// TwinCAT 3 PLC project ICPPLC
// ProgramVersion: 3.1.4023.0
// CompilerDefines: VISU_USEWSTRING
// libraries:
//   Tc2_Math, * (Beckhoff Automation GmbH)
//   Tc2_MC2, * (Beckhoff Automation GmbH)
//   Tc2_SerialCom, * (Beckhoff Automation GmbH)
//   Tc2_Standard, * (Beckhoff Automation GmbH)
//   Tc2_SUPS, * (Beckhoff Automation GmbH)
//   Tc2_System, * (Beckhoff Automation GmbH)
//   Tc2_TcpIp, * (Beckhoff Automation GmbH)
//   Tc2_Utilities, * (Beckhoff Automation GmbH)
//   Tc3_Module, * (Beckhoff Automation GmbH)
//   VisuDialogs, * (System)
//   VisuSymbols, * (System)
// project tree:
//   / ComTask.TcTTO, DataSave_1.TcTTO, GlobalTextList.TcGTLO, IOTask.TcTTO, PlcTask.TcTTO, VISU_TASK.TcTTO, 视图管理器.TcVMO (not stored)
//   DUTs/ ST_A2BData.TcDUT, ST_B2AData.TcDUT
//   GVLs/ GVL_AllCONSTANT.TcGVL, GVL_AllGLOBAL.TcGVL, GVL_AllPERSISTENT.TcGVL, GVL_Datasave.TcGVL
//   POUs/BaseModule/ActionModule/ARMModule/ ARMModule.TcPOU
//   POUs/BaseModule/ActionModule/ARMModule/enum/ ARMType.TcDUT
//   POUs/BaseModule/ActionModule/ARMModule/struct/ ARMModuleHMI.TcDUT
//   POUs/BaseModule/ActionModule/cylinderModule/ CylinderModule.TcPOU
//   POUs/BaseModule/ActionModule/cylinderModule/enum/ CylinderType.TcDUT
//   POUs/BaseModule/ActionModule/cylinderModule/struct/ cylinderModuleHMI.TcDUT
//   POUs/BaseModule/ActionModule/cylinderModule/visu/ cylinderModuleVisu.TcVIS, cylinderModuleVisu_1.TcVIS
//   POUs/BaseModule/ActionModule/chillerModule/ ChillerModule_1.TcPOU
//   POUs/BaseModule/ActionModule/chillerModule/enum/ chillerType.TcDUT
//   POUs/BaseModule/ActionModule/chillerModule/struct/ chillerModuleHMI.TcDUT
//   POUs/BaseModule/ActionModule/enum/ ControlMode.TcDUT
//   POUs/BaseModule/ActionModule/ GVL_ActionModule.TcGVL
//   POUs/BaseModule/ActionModule/HEATModule/enum/ HEATType.TcDUT
//   POUs/BaseModule/ActionModule/HEATModule/ HeatModule.TcPOU
//   POUs/BaseModule/ActionModule/HEATModule/struct/ HEATModuleHMI.TcDUT
//   POUs/BaseModule/ActionModule/HEATModule/visu/ HeatModuleVisu.TcVIS
//   POUs/BaseModule/ActionModule/MFCModule/enum/ MFCType.TcDUT
//   POUs/BaseModule/ActionModule/MFCModule/ MFCModule.TcPOU
//   POUs/BaseModule/ActionModule/MFCModule/struct/ MFCStruct.TcDUT
//   POUs/BaseModule/ActionModule/motorModule/enum/ MotorHomeMode.TcDUT, MotorType.TcDUT
//   POUs/BaseModule/ActionModule/motorModule/ FB_MotorMovements.TcPOU, MotionModule.TcPOU
//   POUs/BaseModule/ActionModule/motorModule/struct/ motionModuleDataHMI.TcDUT, ST_MotorOutput.TcDUT
//   POUs/BaseModule/ActionModule/motorModule/visu/ motionModuleP1.TcVIS, motionModuleP2.TcVIS, motionModuleP3.TcVIS
//   POUs/BaseModule/ActionModule/OtherModule/ ChillerModule.TcPOU, GaugeViewModule.TcPOU, ChamberGaugeViewModule.TcPOU
//   POUs/BaseModule/ActionModule/PendulumValveModule/enum/ PVControlMOD.TcDUT, PVType.TcDUT
//   POUs/BaseModule/ActionModule/PendulumValveModule/ PVModule.TcPOU
//   POUs/BaseModule/ActionModule/PendulumValveModule/struct/ PVModuleHMI.TcDUT
//   POUs/BaseModule/ActionModule/RFModule/enum/ RFType.TcDUT
//   POUs/BaseModule/ActionModule/RFModule/ RFModule.TcPOU
//   POUs/BaseModule/ActionModule/RFModule/struct/ RFHMIStruts.TcDUT
//   POUs/BaseModule/ActionModule/RFModule_Source/ RFModule_Source.TcPOU
//   POUs/BaseModule/ActionModule/TMPModule/enum/ TMPType.TcDUT
//   POUs/BaseModule/ActionModule/TMPModule/struct/ TMPHMIStruts.TcDUT
//   POUs/BaseModule/ActionModule/TMPModule/ TMPModule.TcPOU
//   POUs/BaseModule/ActionModule/TMPModule/visu/ TMPModuleVisu.TcVIS
//   POUs/BaseModule/ActionModule/VPEModule/enum/ VPEType.TcDUT
//   POUs/BaseModule/ActionModule/VPEModule/struct/ VPEHMIStruts.TcDUT, VPETestStruts530.TcDUT, VPETestStruts540.TcDUT
//   POUs/BaseModule/ActionModule/VPEModule/visu/ VPEModuleVis.TcVIS
//   POUs/BaseModule/ActionModule/VPEModule/ VPEModule.TcPOU
//   POUs/BaseModule/COE/ EcCoeSdo_ForTest.TcPOU, FB_ECCOE_READ_WRITE.TcPOU
//   POUs/BaseModule/Communication/ FuncModule_RS232_Byte.TcPOU, FuncModule_RS232_SRF.TcPOU, FuncModule_RS232_ARM.TcPOU, FuncModule_RS485_MFC.TcPOU, FuncModule_RS232_TBP.TcPOU, FuncModule_TCPIP_Binary_POU.TcPOU, FuncModule_TCPIP_String_POU.TcPOU
//   POUs/BaseModule/Communication/struct/ struct_byte_1.TcDUT, struct_Tester.TcDUT, struct_byte.TcDUT
//   POUs/BaseModule/DataSaveModule_EX/csvReadWriteInTextMode/ P_TextModeDelete_1.TcPOU, P_TextModeRead.TcPOU, P_TextModeRead_Recipe.TcPOU, P_TextModeRead_RecipeName.TcPOU, P_TextModeWrite.TcPOU, P_TextModeWrite_Recipe.TcPOU, P_TextModeWrite_RecipeName.TcPOU, StringModel_256000_EX.TcPOU
//   POUs/BaseModule/DataSaveModule_EX/ DataSaveModule_EX.TcPOU, GVL_DataSave_EX.TcGVL, RecipeNameModule_EX.TcPOU, RecipeSaveModule_EX.TcPOU
//   POUs/BaseModule/DataSaveModule_EX/Struct/ RecipeNamePar.TcDUT, RecipePar.TcDUT, RecipeShowStr.TcDUT
//   POUs/BaseModule/EL2252_2262Control/ FlipperModule_EL2252.TcPOU, FlipperModule_EL2262.TcPOU, FlipperModule_EL2262_old.TcPOU
//   POUs/BaseModule/EL2252_2262Control/SquareWaveOut/ FB_SquareWaveOut_EL2262.TcPOU, SquareWaveOut_EL2262_TEST.TcPOU
//   POUs/BaseModule/EL2252_2262Control/struct/ ST_CamSwitch.TcDUT, ST_CamSwitch_EL2262.TcDUT, ST_EL2262OutData.TcDUT
//   POUs/BaseModule/Error/enum/ Error_Level.TcDUT
//   POUs/BaseModule/Error/ ErrCodeProcess.TcPOU, errorMonitor.TcPOU, error_Printf.TcPOU, error_Trigger.TcPOU, GVL_Error.TcGVL
//   POUs/BaseModule/Error/struct/ ST_Error.TcDUT
//   POUs/BaseModule/IO/ FB_IOBase_Input_New.TcPOU, FB_IOBase_Output_New.TcPOU
//   POUs/BaseModule/IO/ReadWriteCSV/ FB_IOFileReadWrite.TcPOU, POU_Test.TcPOU, ST_DataFmtBase.TcDUT
//   POUs/BaseModule/IO/struct/ ST_INPUT_IO.TcDUT, ST_IOBase_Show_HMI.TcDUT, ST_OUTPUT_IO.TcDUT
//   POUs/BaseModule/IO/visu/ IOBase_Show_New.TcVIS
//   POUs/BaseModule/MainFrame/ MainFram.TcDUT, MainFrame.TcVIS
//   POUs/BaseModule/PrintLogModule_EX/ GVL_PrintLogModule_EX.TcGVL, printLogModule_EX.TcPOU
//   POUs/BaseModule/PrintLogModule_EX/struct/ printLogModule_EX_DataHMI.TcDUT, printLogModule_EX_DataST.TcDUT, ST_DeleteFile.TcDUT
//   POUs/BaseModule/PrintLogModule_EX/visu/ showInfo_Auto.TcVIS, showInfo.TcVIS
//   POUs/BaseModule/SystemTimeModule/ GVL_SystemTimeModule.TcGVL, systemTimeModule.TcPOU
//   POUs/BaseModule/TcpIpModule_EX/ ALCData2String.TcPOU, CloseAllSocket.TcPOU, GVL_TcpIpModule_EX.TcGVL
//   POUs/BaseModule/TcpIpModule_EX/clientModule_EX/ tcpipClientModule_EX.TcPOU
//   POUs/BaseModule/TcpIpModule_EX/dataStruct_EX/ ST_TCPIP_DATA_STRUCT_ALC.TcDUT
//   POUs/BaseModule/TcpIpModule_EX/serverModule_EX/ tcpipServerModule_EX.TcPOU
//   POUs/BaseModule/UPS_CX51X0/ ups_CX51X0.TcPOU
//   POUs/Communication/ Communication_Error.TcPOU, PLC_Chiller.TcPOU, PLC_AMX_AI.TcPOU, PLC_FreeByte.TcPOU, PLC_PDV.TcPOU, PLC_HeliumPressure.TcPOU, PLC_SourceRF.TcPOU, PLC_PowerRF.TcPOU, PRG_ADS_Comm_ByName_A2B.TcPOU, RS232_485_ALLEL.TcPOU, PLC_String.TcPOU, PLC_SW1.TcPOU, ServicesRefreshPOU.TcPOU
//   POUs/Communication/Communica_ALC/ enum_CommandNumber.TcDUT, E_Sta1_CMD.TcDUT
//   POUs/Data/ DataSave.TcPOU, DownTimeRecordPOU.TcPOU, FB_SavePar.TcPOU, FB_WStringSave.TcPOU, Test_FilePOU.TcPOU
//   POUs/Instance/ instance.TcPOU, InstanceUtility.TcPOU
//   POUs/IO/ TesterIO.TcPOU
//   POUs/MachinePOU/SemiAutomatic/ S_BackOfHeliumClear.TcPOU, S_CO_ControlRF.TcPOU, S_PDVSafeCtr.TcPOU, S_MachineVent.TcPOU, S_Etching.TcPOU, S_LoadLockPumping.TcPOU, S_LoadLockVent.TcPOU, S_ChamberLLVent.TcPOU, S_MachinePumping.TcPOU, S_UnLoadWafer.TcPOU, S_WaferCheckPOU.TcPOU, S_RoughPumping.TcPOU, S_ActuatorRecoveryPOU.TcPOU, S_LoadWafer.TcPOU
//   POUs/MachinePOU/State/ otherMachineState.TcPOU
//   POUs/MachinePOU/ MainPOU.TcPOU
//   POUs/ MAIN.TcPOU
//   POUs/Other/ActBase/ ActStepBase.TcPOU
//   POUs/Other/ActBase/ITF/ ITFActStep.TcIO, ITFUserAction.TcIO
//   POUs/Other/ActBase/ITF/struct/ ST_ActStep_State.TcDUT
//   POUs/Other/HMI/ Note.TcVIS, WARMStruct.TcDUT, WARM.TcVIS, NoteStruct.TcDUT
//   POUs/Other/MachineState/enum/ RunningStatus.TcDUT
//   POUs/Other/MachineState/ FB_MachineState.TcPOU, GVL_MachineState.TcGVL, MachineStatePOU.TcPOU, MainParComfer_HMI.TcPOU, ST_DownTimeRecord.TcDUT, ST_MachineState.TcDUT
//   POUs/Other/ MainRunPOU.TcPOU
//   POUs/Other/Struct/ActPos/ ST_DOEActPos.TcDUT
//   POUs/Other/Struct/StationBuild/ ST_ICP.TcDUT
//   POUs/Other/Struct/ ST_HaveDUTState.TcDUT, ST_MachineUtility.TcDUT, ST_POUCommunication.TcDUT, ST_StationConfigBase.TcDUT
//   VISUs/Editor/ Manual.TcVIS, Overview.TcVIS, Overview_Total.TcVIS, ViewPar.TcVIS, ViewPar_1.TcVIS
//   VISUs/Config/ Config.TcVIS, Config_Base.TcVIS
//   VISUs/ ImagePool1.TcIPO (not stored), Loadding.TcVIS, Main.TcVIS
//   VISUs/IO/ IO.TcVIS, IO_Input.TcVIS, IO_Output.TcVIS
//   VISUs/Log/ LogInf.TcVIS
//   VISUs/Operator/ Operator.TcVIS
//   VISUs/Recipe/ Recipe.TcVIS, Recipe_Operator.TcVIS
//   VISUs/TextList/ CtrlModeTextList.TcTLO, MachineStateTextList.TcTLO, PDVConfigMode.TcTLO, RunModeTypeTexList.TcTLO
// real-time tasks:
//   TASK PlcTask: cycle T#10ms, priority 17, ADS port 350
//   TASK VISU_TASK: cycle T#100000us, priority 30, ADS port 351
//   TASK DataSave_1: cycle T#20ms, priority 18, ADS port 352
//   TASK IOTask: cycle T#2ms, priority 12, ADS port 353
//   TASK ComTask: cycle T#2ms, priority 19, ADS port 354
// I/O:
//   DEVICE Device 1 (EtherCAT), AmsNetId 5.114.113.208.2.1
//     Term 1 (EK1200) [EK1200-5000 EtherCAT Power supply (2A E-Bus)]
//       Term 2 (EL1889) [EL1889 16Ch. Dig. Input 24V, 3ms, negative]
//       Term 3 (EL1889) [EL1889 16Ch. Dig. Input 24V, 3ms, negative]
//       Term 4 (EL2889) [EL2889 16Ch. Dig. Output 24V, 0.5A, negative]
//       Term 5 (EL2889) [EL2889 16Ch. Dig. Output 24V, 0.5A, negative]
//       Term 6 (EL2889) [EL2889 16Ch. Dig. Output 24V, 0.5A, negative]
//       Term 7 (EL3174) [EL3174 4K. Ana. Eingang  +/-10V Diff., +/-20mA SingleEnded, 16 Bit]
//       Term 8 (EL6002) [EL6002 Interface 2Ch. (RS232)]
//       Term 9 (EL6002) [EL6002 Interface 2Ch. (RS232)]
//       Term 10 (EL6022) [EL6022 Interface 2Ch. (RS422/485)]
//       Term 11 (EK1110) [EK1110 EtherCAT extension]
//   DEVICE Device 6 (EtherCAT), AmsNetId 5.114.113.208.7.1
//     Box 12 (EC SERIES) [EC SERIES]
// variable links:
//   ICPPLC/ICPPLC Instance <-> Device 1 (EtherCAT)/Term 1 (EK1200)/Term 10 (EL6022)
//     ComTask Inputs/RS232_485_ALLEL.MFC_COMin/D[{0..21}] <-> COM Inputs Channel 2/Data In {0..21}  (22 links)
//     ComTask Inputs/RS232_485_ALLEL.MFC_COMin/Status <-> COM Inputs Channel 2/Status
//     ComTask Outputs/RS232_485_ALLEL.MFC_COMout/Ctrl <-> COM Outputs Channel 2/Ctrl
//     ComTask Outputs/RS232_485_ALLEL.MFC_COMout/D[{0..21}] <-> COM Outputs Channel 2/Data Out {0..21}  (22 links)
//   ICPPLC/ICPPLC Instance <-> Device 1 (EtherCAT)/Term 1 (EK1200)/Term 2 (EL1889)
//     IOTask Inputs/TesterIO.fbIOBase_Input.stIOBase[1].io[{1..16}] <-> Channel {1..16}/Input  (16 links)
//   ICPPLC/ICPPLC Instance <-> Device 1 (EtherCAT)/Term 1 (EK1200)/Term 3 (EL1889)
//     IOTask Inputs/TesterIO.fbIOBase_Input.stIOBase[2].io[{1..16}] <-> Channel {1..16}/Input  (16 links)
//   ICPPLC/ICPPLC Instance <-> Device 1 (EtherCAT)/Term 1 (EK1200)/Term 4 (EL2889)
//     IOTask Outputs/TesterIO.fbIOBase_Output.stIOBase[1].io[{1..16}] <-> Channel {1..16}/Output  (16 links)
//   ICPPLC/ICPPLC Instance <-> Device 1 (EtherCAT)/Term 1 (EK1200)/Term 5 (EL2889)
//     IOTask Outputs/TesterIO.fbIOBase_Output.stIOBase[2].io[{1..16}] <-> Channel {1..16}/Output  (16 links)
//   ICPPLC/ICPPLC Instance <-> Device 1 (EtherCAT)/Term 1 (EK1200)/Term 6 (EL2889)
//     IOTask Outputs/TesterIO.fbIOBase_Output.stIOBase[3].io[{1..16}] <-> Channel {1..16}/Output  (16 links)
//   ICPPLC/ICPPLC Instance <-> Device 1 (EtherCAT)/Term 1 (EK1200)/Term 7 (EL3174)
//     PlcTask Inputs/GVL_AllGLOBAL.gICP.AI_AIMGauge <-> AI Standard Channel 2/Value
//     PlcTask Inputs/GVL_AllGLOBAL.gICP.AI_ChamberGauge <-> AI Standard Channel 4/Value
//     PlcTask Inputs/GVL_AllGLOBAL.gICP.AI_ForeLineGauge <-> AI Standard Channel 1/Value
//     PlcTask Inputs/GVL_AllGLOBAL.gICP.AI_LoadLockGauge <-> AI Standard Channel 3/Value
//   ICPPLC/ICPPLC Instance <-> Device 1 (EtherCAT)/Term 1 (EK1200)/Term 9 (EL6002)
//     ComTask Inputs/RS232_485_ALLEL.ARM_COMin/D[{0..21}] <-> COM TxPDO-Map Inputs Channel 1/Data In {0..21}  (22 links)
//     ComTask Inputs/RS232_485_ALLEL.ARM_COMin/Status <-> COM TxPDO-Map Inputs Channel 1/Status
//     ComTask Inputs/RS232_485_ALLEL.TBP_COMin/D[{0..21}] <-> COM TxPDO-Map Inputs Channel 2/Data In {0..21}  (22 links)
//     ComTask Inputs/RS232_485_ALLEL.TBP_COMin/Status <-> COM TxPDO-Map Inputs Channel 2/Status
//     ComTask Outputs/RS232_485_ALLEL.ARM_COMout/Ctrl <-> COM RxPDO-Map Outputs Channel 1/Ctrl
//     ComTask Outputs/RS232_485_ALLEL.ARM_COMout/D[{0..21}] <-> COM RxPDO-Map Outputs Channel 1/Data Out {0..21}  (22 links)
//     ComTask Outputs/RS232_485_ALLEL.TBP_COMout/Ctrl <-> COM RxPDO-Map Outputs Channel 2/Ctrl
//     ComTask Outputs/RS232_485_ALLEL.TBP_COMout/D[{0..21}] <-> COM RxPDO-Map Outputs Channel 2/Data Out {0..21}  (22 links)
//   ICPPLC/ICPPLC Instance <-> Device 6 (EtherCAT)/Box 12 (EC SERIES)
//     PlcTask Inputs/GVL_AllGLOBAL.gICP.HeMFC_ActFlow <-> SDP TxPDO Map/Flow Reading
//     PlcTask Outputs/GVL_AllGLOBAL.gICP.HeMFC_SetFlow <-> SDP RxPDO Map/Flow SP

CONFIGURATION ICPPLC
    RESOURCE PLC ON TwinCAT3
        TASK ComTask(INTERVAL := T#2ms, PRIORITY := 19);
        TASK DataSave_1(INTERVAL := T#20ms, PRIORITY := 18);
        TASK IOTask(INTERVAL := T#2ms, PRIORITY := 12);
        TASK PlcTask(INTERVAL := T#10ms, PRIORITY := 17);
        TASK VISU_TASK(INTERVAL := T#100000us, PRIORITY := 30);
        PROGRAM RS232_485_ALLEL WITH ComTask : RS232_485_ALLEL;
        PROGRAM DataSave WITH DataSave_1 : DataSave;
        PROGRAM TesterIO WITH IOTask : TesterIO;
        PROGRAM MAIN WITH PlcTask : MAIN;
        PROGRAM VisuElems_Visu_Prg WITH VISU_TASK : VisuElems.Visu_Prg;
    END_RESOURCE
END_CONFIGURATION

// ---- DUTs/ST_A2BData.TcDUT
TYPE ST_A2BData :// 主控(Gideon)给新松
STRUCT
	bRunning					:BOOL;// 允许标志
	bError						:BOOL;// 报错
	bHeartBeatMonitor			:BOOL;// 心跳监控
	// 命令
	Cmd_1						:BOOL; 	
	Cmd_2						:BOOL; 	
	Cmd_3						:BOOL; 
	Cmd_4						:BOOL; 
	Cmd_5						:BOOL; 	
	Cmd_6						:BOOL; 	
	Cmd_7						:BOOL; 	
	Cmd_8						:BOOL; 
	Cmd_9						:BOOL; 
	Cmd_10						:BOOL;		
	// 反馈
	O_1							:BOOL;   
	O_2							:BOOL;
	O_3							:BOOL;
	O_4							:BOOL;                                  
	O_5							:BOOL;
	O_6							:BOOL;
	O_7							:BOOL;
	O_8							:BOOL;
	O_9							:BOOL;
	O_10						:BOOL;
	// 回传
	I_1							:BOOL;   
	I_2							:BOOL;
	I_3							:BOOL;
	I_4							:BOOL;                                  
	I_5							:BOOL;
	I_6							:BOOL;
	I_7							:BOOL;
	I_8							:BOOL;
	I_9							:BOOL;
	I_10						:BOOL;
END_STRUCT
END_TYPE

// ---- DUTs/ST_B2AData.TcDUT
TYPE ST_B2AData :// 主控(Gideon)给新松
STRUCT
	bRunning					:BOOL;// 允许标志
	bError						:BOOL;// 报错
	bHeartBeatMonitor			:BOOL;// 心跳监控
	// 命令
	Sub_1						:BOOL; 	
	Sub_2						:BOOL; 	
	Sub_3						:BOOL; 
	Sub_4						:BOOL; 
	Sub_5						:BOOL; 	
	Sub_6						:BOOL; 	
	Sub_7						:BOOL; 	
	Sub_8						:BOOL; 
	Sub_9						:BOOL; 
	Sub_10						:BOOL;		
	// 反馈
	O_1							:BOOL;   
	O_2							:BOOL;
	O_3							:BOOL;
	O_4							:BOOL;                                  
	O_5							:BOOL;
	O_6							:BOOL;
	O_7							:BOOL;
	O_8							:BOOL;
	O_9							:BOOL;
	O_10						:BOOL;
	// 回传
	I_1							:BOOL;   
	I_2							:BOOL;
	I_3							:BOOL;
	I_4							:BOOL;                                  
	I_5							:BOOL;
	I_6							:BOOL;
	I_7							:BOOL;
	I_8							:BOOL;
	I_9							:BOOL;
	I_10						:BOOL;
END_STRUCT
END_TYPE

// ---- POUs/BaseModule/ActionModule/ARMModule/enum/ARMType.TcDUT

TYPE ARMType :
(
	ARMType_Default := 0, //常规的ARM
	ARMType_SinSun := 1, // 新松
	ARMType_Other := 2 // 蝶阀
)UINT;
END_TYPE

// ---- POUs/BaseModule/ActionModule/ARMModule/struct/ARMModuleHMI.TcDUT
{attribute 'pack_mode' := 1}
TYPE ARMModuleHMI :
STRUCT
//control signal or data
	INAndHOME		: BOOL:=FALSE;// 单控件触发信号

	IN				: BOOL:=FALSE;// IN触发信号
	HOME			: BOOL:=FALSE;// HOME触发信号
	reset			: BOOL:=FALSE;// 复位信号
	stop			: BOOL:=FALSE;// 停止信号
	power			: BOOL:=TRUE;//no power, two relay will lost power

//monitor
	INAprSw			: BOOL:=FALSE;//HW: ARM IN approach switch
	HOMEAprSw		: BOOL:=FALSE;//HW: ARM HOME approach switch	
	INRelay			: BOOL:=FALSE;//HW: ARM IN action relay
	HOMERelay		: BOOL:=FALSE;//HW: ARM HOME action relay	

	enableHome		: BOOL:=TRUE;//for outside control instance
	enableIN		: BOOL:=TRUE;//for outside control instance
//state
	HMIEnable		: BOOL:=TRUE;
	enable			: BOOL;
	busy			: BOOL;
	done			: BOOL;
	error			: BOOL;
	extenderror		: BOOL;
	retracterror	: BOOL;
	errID			: DINT;
	nameTXT			: STRING;// ARM名字
	errTXT			: STRING;
	INcondition		: BOOL;// IN条件
	HOMEcondition	: BOOL;// HOME条件
END_STRUCT
END_TYPE
(*
按照字节对齐规则，将变量按字节大小按顺序定义，用于ADS读取
*)

// ---- POUs/BaseModule/ActionModule/cylinderModule/enum/CylinderType.TcDUT

TYPE CylinderType :
(
	CylinderType_Default := 0, //常规的气缸
	CylinderType_Vacuum := 1, //真空发生器
	CylinderType_ButV := 2 // GateDoor
)UINT;
END_TYPE

// ---- POUs/BaseModule/ActionModule/cylinderModule/struct/cylinderModuleHMI.TcDUT
{attribute 'pack_mode' := 1}
TYPE cylinderModuleHMI :
STRUCT
//control signal or data
	extendAndretract: BOOL:=FALSE;//单控件触发信号
	singleControl	: BOOL:=FALSE;//单一信号控制
	singleControltemp: BOOL:=FALSE;//单一信号控制
	extend			: BOOL:=FALSE;//伸出触发信号
	retract			: BOOL:=FALSE;//收回触发信号
	reset			: BOOL:=FALSE;//复位信号
	stop			: BOOL:=FALSE;//停止信号
	power			: BOOL:=TRUE;//no power, two relay will lost power
	showWarm		: BOOL:=FALSE;// show warm txt
//monitor
	extAprSw		: BOOL:=FALSE;//HW: cylinder extent approach switch
	retAprSw		: BOOL:=FALSE;//HW: cylinder retract approach switch	
	extRelay		: BOOL:=FALSE;//HW: cylinder extent action relay
	retRelay		: BOOL:=FALSE;//HW: cylinder retract action relay	

	enableExt		: BOOL:=TRUE;//for outside control instance
	enableRet		: BOOL:=TRUE;//for outside control instance
//state
	HMIEnable		: BOOL:=TRUE;
	enable			: BOOL;
	busy			: BOOL;
	done			: BOOL;
	error			: BOOL;
	extenderror		: BOOL;
	retracterror	: BOOL;
	errID			: DINT;
	nameTXT			: STRING;//气缸名字
	errTXT			: STRING;
	sensorShow		: STRING;
	extcondition	: BOOL;// 开条件
	retcondition	: BOOL;// 关条件
END_STRUCT
END_TYPE
(*
按照字节对齐规则，将变量按字节大小按顺序定义，用于ADS读取
*)

// ---- POUs/BaseModule/ActionModule/chillerModule/enum/chillerType.TcDUT

TYPE chillerType :
(
	ChillerType_Default := 0, //常规水冷机
	ChillerType_Vacuum := 1, // 未知1
	ChillerType_ButV := 2 // 未知1
)UINT;
END_TYPE

// ---- POUs/BaseModule/ActionModule/chillerModule/struct/chillerModuleHMI.TcDUT
{attribute 'pack_mode' := 1}
TYPE chillerModuleHMI :
STRUCT
//control signal or data
	extendAndretract: BOOL:=FALSE;//单控件触发信号
	singleControl	: BOOL:=FALSE;//单一信号控制
	singleControltemp: BOOL:=FALSE;//单一信号控制
	extend			: BOOL:=FALSE;//伸出触发信号
	retract			: BOOL:=FALSE;//收回触发信号
	reset			: BOOL:=FALSE;//复位信号
	stop			: BOOL:=FALSE;//停止信号
	set				: BOOL:=false;// 参数设定
	power			: BOOL:=TRUE;//no power, two relay will lost power
	setpointVal		:REAL;
//monitor
	extAprSw		: BOOL:=FALSE;//HW: cylinder extent approach switch
	retAprSw		: BOOL:=FALSE;//HW: cylinder retract approach switch	
	extRelay		: BOOL:=FALSE;//HW: cylinder extent action relay
	retRelay		: BOOL:=FALSE;//HW: cylinder retract action relay	

	enableExt		: BOOL:=TRUE;//for outside control instance
	enableRet		: BOOL:=TRUE;//for outside control instance
//state
	HMIEnable		: BOOL:=TRUE;
	enable			: BOOL;
	busy			: BOOL;
	done			: BOOL;
	error			: BOOL;
	extenderror		: BOOL;
	retracterror	: BOOL;
	errID			: DINT;
	nameTXT			: STRING;//气缸名字
	errTXT			: STRING;
	sensorShow		: STRING;
	extcondition	: BOOL;// 开条件
	retcondition	: BOOL;// 关条件
END_STRUCT
END_TYPE
(*
按照字节对齐规则，将变量按字节大小按顺序定义，用于ADS读取
*)

// ---- POUs/BaseModule/ActionModule/enum/ControlMode.TcDUT
TYPE ControlMode :
(
	eAutoCtrMode	 	:= 1,//自动控制模式
	eManualCtrMode		:= 2,//手动控制模式
	eDebugMode			:= 3,//待开发
	eSemiAutoMode		:= 4,//半自动控制模式
	
	eLoopMode			:= 8,//老化模式
	eConfig				:= 9//配置模式
)UINT;
END_TYPE

// ---- POUs/BaseModule/ActionModule/HEATModule/enum/HEATType.TcDUT
TYPE HEATType :
(
	HEATType_Default := 0, // 常规的加热,两者都具备
	HEATType_Smart := 1, // 智能加热
	HEATType_Manul := 2 // 手动加热
)UINT;
END_TYPE

// ---- POUs/BaseModule/ActionModule/HEATModule/struct/HEATModuleHMI.TcDUT
{attribute 'pack_mode' := 1}
TYPE HEATModuleHMI :
STRUCT
	// Aiko
	bHeat			:BOOL:=FALSE;// 加热停止一个按钮，根据状态决定是否加热等操作
	oheatStart		:BOOL;// 加热输出
	iheatStart		:BOOL;// 加热反馈
//control signal or data
	heat			: BOOL:=FALSE;// 加热中
	ATLearning		: BOOL:=FALSE;// 参数自学习
	manuleHeat		: BOOL:=FALSE;// 手动加热
	reset			: BOOL:=FALSE;// 复位信号
	stop			: BOOL:=FALSE;// 停止信号
	power			: BOOL:=TRUE;//  no power, two relay will lost power

//monitor	
	status_PV			:REAL;// 温控反馈测量值
	status_MV			:INT;// 温控反馈Manul设定值
	status_P			:INT;// 温控反馈P参数
	status_I			:INT;// 温控反馈I参数
	status_D			:REAL;// 温控反馈D参数
	
	heatDoneCheckMaxTime:DINT:=300;// 加热完成检测超时时间,单位秒S
//state
	ctrl_heatStart		: BOOL;//bit0 开始加热
	ctrl_heatATStart	: BOOL;//bit2 100%AT实行中
	ctrl_heatATStop		: BOOL;//bit4 AT取消
	ctrl_heatAuto		: BOOL;//bit5 0: Auto,1: Manul
	
	para_Manual_MV		:INT;// 手动MV
	para_SV				:REAL;// 温度设定值
	para_P				:INT;// 温控P参数
	para_I				:INT;// 温控I参数
	para_D				:REAL;// 温控D参数
	para_HLimit			:REAL;// 温控报警上限参数
	para_LLimit			:REAL;// 温控报警下限参数
	
	para_setTOffset		:REAL:=1.0;// 温控偏差
	
	HMIEnable		: BOOL:=TRUE;
	busy			: BOOL;// 加热中 
	done			: BOOL;
	error			: BOOL;
	errID			: DINT;
	nameTXT			: STRING;
	errTXT			: STRING;
END_STRUCT
END_TYPE
(*
按照字节对齐规则，将变量按字节大小按顺序定义，用于ADS读取
*)

// ---- POUs/BaseModule/ActionModule/MFCModule/enum/MFCType.TcDUT
TYPE MFCType :
(
	MFCType_Default := 0 //常规分子MFC
)UINT;
END_TYPE

// ---- POUs/BaseModule/ActionModule/MFCModule/struct/MFCStruct.TcDUT
{attribute 'pack_mode' := 1}
TYPE MFCStruct :
STRUCT
	set:BOOL;
	clear:BOOL;
END_STRUCT
END_TYPE
(*
按照字节对齐规则，将变量按字节大小按顺序定义，用于ADS读取
*)

// ---- POUs/BaseModule/ActionModule/motorModule/enum/MotorHomeMode.TcDUT
TYPE MotorHomeMode :
(
	MotorHomeMode_Default	 				:= 0, 	//电机Home模式 默认有正负限位/原点信号
	MotorHomeMode_PLimitSwitch_To_DOG 		:= 1,	//电机Home模式 正限位做零点信号
	MotorHomeMode_NLimitSwitch_To_DOG		:= 2,	//电机Home模式 负限位做零点信号
	MotorHomeMode_OnlyDOGPointSwitch		:= 3	//电机Home模式 只有原点信号, 执行往复搜寻动作
)UINT;
END_TYPE

// ---- POUs/BaseModule/ActionModule/motorModule/enum/MotorType.TcDUT
TYPE MotorType :
(
	MotorType_Default	 	:= 0, 		//增量式编码器(需要执行McHome)
	MotorType_DDmotor_HC 	:= 1,		//横川DD马达(不需要执行McHome,使用高创驱动器自带的回原点方式)
	MotorType_Absolute		:= 2		//绝对式编码器(不需要执行McHome)
)UINT;
END_TYPE

// ---- POUs/BaseModule/ActionModule/motorModule/struct/motionModuleDataHMI.TcDUT
{attribute 'pack_mode' := 1}
TYPE motionModuleDataHMI :
STRUCT
//************************* control *************************	
 //button
 	// Aiko
	manJogN					: BOOL:=FALSE;
	manJogP					: BOOL:=FALSE;
	manVelN					: BOOL:=FALSE;
	manVelP					: BOOL:=FALSE;
	GoToOpen				: BOOL:=FALSE;// 去开门位
	GoToClose				: BOOL:=FALSE;// 去关门位
	// normal 
	manJogGo				: BOOL:=FALSE;
	manRelGo				: BOOL:=FALSE;
	manVelGo				: BOOL:=FALSE;
	manABSGo				: BOOL:=FALSE;
	reset					: BOOL;
	stop					: BOOL;
	choiceOfDirection		: BOOL:=TRUE;
	setZero					: BOOL:=FALSE;
	power					: BOOL:=TRUE;
	goHomeGo				: BOOL:=FALSE;
	pauseB					: BOOL;
	loopRelGo				: BOOL:=FALSE;//loop 相对运动启动
	loopAbsGo				: BOOL:=FALSE;//loop 绝对运动启动
	loopHomeToPosGo			: BOOL:=FALSE;//loop 循环回原到指定点位打表
	
 //monitor status
	forwardLimitSwitch		: BOOL;//正限位感应 状态
	backwardsLimitSwitch	: BOOL;//负限位感应 状态
	dogPointSwitch			: BOOL;//原点感应 状态
	forwardEnable			: BOOL;//正限位启用/禁用 状态
	backwardsEnable			: BOOL;//负限位启用/禁用 状态
	busy					: BOOL;//busy 状态
	done					: BOOL;//done 状态
	error					: BOOL;//error 状态
	oPause					: BOOL;//pause 状态
	powerEnable				: BOOL;//使能启用/禁用 
	enable					: BOOL;//enable 状态
	goHomeDone				: BOOL;//Home 完成状态
	running					: BOOL;// 运行状态
	jogNrunning				: BOOL;// Jog反向运行状态
	jogPrunning				: BOOL;// Jog反向运行状态
	velNrunning				: BOOL;// vel反向运行状态
	velPrunning				: BOOL;// vel反向运行状态
	
 //
	ctrlModeCondition		: BOOL;// 手动控制条件
	jogCondition			: BOOL;// JOG 可触发条件
	velCondition			: BOOL;// 速度模式定位 可触发条件
	relCondition			: BOOL;// 相对定位 可触发条件
	absCondition			: BOOL;// 绝对定位 可触发条件
	homeCondition			: BOOL;// Home 可触发条件
	setCondition			: BOOL;// 目标位置设定 可触发条件
	loopRelCondition		: BOOL;// loop相对定位 可触发条件
	loopAbsCondition		: BOOL;// loop绝对定位 可触发条件
	loopHomeToAbsCondition	: BOOL;// loop绝对定位 回原 可触发条件
	
//************************* para *************************
	loopCycle				: UINT:=0;//loop 循环次数 一次往复才算一次
	loopWatingTime			: UINT:=1000;//loop 停留时间（单位ms）
	errID					: DINT;//errorID
	PTPErrID				: UDINT;//PTPErrID

	manABSPos				: LREAL:=0;	//ABS target position
	manRelDis				: LREAL:=0;	//REL target distance
	manVel					: LREAL:=3;//abs, rel use the same one value
	manJogVel				: LREAL:=1;	//jog, vel use the same one value
	actualPos				: LREAL;//actual pos
	actualVel				: LREAL;//actual vel
	goHomeVel				: LREAL:=10;
	goHomeVelSlow			: LREAL:=5;
	softPLimitPos			: LREAL:=99999999999;
	softNLimitPos			: LREAL:=-99999999999;
	loopFirstPoint			: LREAL:=0;//loop 第1个点
	loopSecondPoint			: LREAL:=0;//loop 第2个点
	loopGoVel				: LREAL:=10;//loop 运动速率
	
	nameTXT					: STRING;//电机名字
	errTxt					: STRING;
	errWTxt					: WSTRING;
	
	GoToOpenDone			: BOOL:=FALSE;// 去开门位
	GoToCloseDone			: BOOL:=FALSE;// 去关门位
//Velo Limit
	manSoftLimitVel			:LREAL:=5.0;// 速度限制
END_STRUCT
END_TYPE
(*
按照字节对齐规则，将变量按字节大小按顺序定义，用于ADS读取
*)

// ---- POUs/BaseModule/ActionModule/motorModule/struct/ST_MotorOutput.TcDUT
{attribute 'pack mode' := 1}
TYPE ST_MotorOutput :
STRUCT
	axisPause						:BOOL;//轴的Pause状态
	axisBusy						:BOOL;//轴的Busy状态
	axisDone						:BOOL;//轴的Done状态
	axisError						:BOOL;//轴的Error状态
	axisHomeState					:BOOL:=FALSE;//轴的原点状态
	
	jogCondition					:BOOL;//轴JOG运动启动条件
	absCondition					:BOOL;//轴绝对运动启动条件
	relCondition					:BOOL;//轴相对运动启动条件
	velCondition					:BOOL;//轴速度模式启动条件
	homeCondition					:BOOL;//轴go home的启动条件
	setCondition					:BOOL;//轴当前位置设定启动条件
	moveModuloCondition				:BOOL;//轴模运动启动条件
	
	axisErrId						:UDINT;//轴的Error Id值
	axisActualPos					:LREAL:=0;//轴的实际位置
	axisActualVel					:LREAL:=0;//轴的实际速率
	axisActualtorque				:LREAL:=0;//轴的实际扭力
	axisErrTxt						:STRING;//轴的报错文本信息
	axisErrWTxt						:WSTRING;//轴的报错文本信息 中文
	
	pAxis	  						:POINTER TO AXIS_REF;
	pMotionModule					:POINTER TO MotionModule;
END_STRUCT
END_TYPE

// ---- POUs/BaseModule/ActionModule/PendulumValveModule/enum/PVControlMOD.TcDUT

TYPE PVControlMOD :
(
	PVControl_Default := 0, // 位置控制
	PVControl_Pressure := 1, // 压力控制模式
	PVControl_Other := 2 // Other
)UINT;
END_TYPE

// ---- POUs/BaseModule/ActionModule/PendulumValveModule/enum/PVType.TcDUT

TYPE PVType :
(
	PVType_Default := 0, // 常规的PV阀
	PVType_VAT := 1, // VAT
	PVType_Other := 2 // Other
)UINT;
END_TYPE

// ---- POUs/BaseModule/ActionModule/PendulumValveModule/struct/PVModuleHMI.TcDUT
{attribute 'pack_mode' := 1}
TYPE PVModuleHMI :
STRUCT
//control signal or data
	OpenAndClose	: BOOL:=FALSE;//单控件触发信号

	open			: BOOL:=FALSE;//打开触发信号
	close			: BOOL:=FALSE;//关闭触发信号
	opentemp		: BOOL:=FALSE;//打开触发信号
	closetemp		: BOOL:=FALSE;//关闭触发信号
	reset			: BOOL:=FALSE;//复位信号
	stop			: BOOL:=FALSE;//停止信号
	power			: BOOL:=TRUE;//no power, two relay will lost power
	
	mode			: BOOL:=FALSE; // 控制模式 false Pos;true PRE
	modetemp		: BOOL:=FALSE; // 控制模式 false Pos;true PRE
	
	set				: BOOL;
	clear			: BOOL;		
	config			: BOOL;		
	
	setPressure		: REAL:=0.0;// 压力值
	setflag			: BOOL;
	clearflag		: BOOL;
	actPressure		: REAL:=0.0;// 实际压力值
	actPos			: REAL:=0.0;// 实际开度

//monitor
	openAprSw		: BOOL:=FALSE;//HW: PV openent approach switch
	closeAprSw		: BOOL:=FALSE;//HW: PV close approach switch	
	openRelay		: BOOL:=FALSE;//HW: PV openent action relay
	closeRelay		: BOOL:=FALSE;//HW: PV close action relay	

	enableopen		: BOOL:=TRUE;//for outside control instance
	enableclose		: BOOL:=TRUE;//for outside control instance
//state
	HMIEnable		: BOOL:=TRUE;
	enable			: BOOL;
	busy			: BOOL;
	done			: BOOL;
	error			: BOOL;
	openerror		: BOOL;
	closeerror		: BOOL;
	errID			: DINT;
	nameTXT			: STRING;// PV名字
	errTXT			: STRING;
	opencondition	: BOOL;// 开条件
	closecondition	: BOOL;// 关条件
	
	setPointNotEq	:BOOL;
END_STRUCT
END_TYPE
(*
按照字节对齐规则，将变量按字节大小按顺序定义，用于ADS读取
*)

// ---- POUs/BaseModule/ActionModule/RFModule/enum/RFType.TcDUT
TYPE RFType :
(
	RFType_Default := 0 //常规分子泵
)UINT;
END_TYPE

// ---- POUs/BaseModule/ActionModule/RFModule/struct/RFHMIStruts.TcDUT
{attribute 'pack_mode' := 1}
TYPE RFHMIStruts :
STRUCT
	// Aiko
	extendAndretract: BOOL:=FALSE;//单控件触发信号
	singleControl	: BOOL:=FALSE;//单一信号控制
	singleControltemp	: BOOL:=FALSE;//单一信号控制
	
	bopen			: BOOL:=FALSE;//启动触发信号
	runTimeClear	: BOOL:=FALSE;//清空计时时间
//control signal or data
	open			: BOOL:=FALSE;//启动触发信号
	close			: BOOL:=FALSE;//停止触发信号
	reset			: BOOL:=FALSE;//复位信号
	stop			: BOOL:=FALSE;//停止信号
	power			: BOOL:=TRUE;//no power, two relay will lost power

//monitor
	AccAprSw		: BOOL:=FALSE;//HW: cylinder extent approach switch
	DccAprSw		: BOOL:=FALSE;//HW: cylinder retract approach switch	
	NormalAprSw		: BOOL:=FALSE;//HW: cylinder retract approach switch	
	AlmAprSw		: BOOL:=FALSE;//HW: cylinder retract approach switch
	ErrorAprSw		: BOOL:=FALSE;//HW: cylinder retract approach switch
	
	openRelay		: BOOL:=FALSE;//HW: cylinder extent action relay
	closeRelay		: BOOL:=FALSE;//HW: cylinder retract action relay	
	resetRelay		: BOOL:=FALSE;//HW: cylinder retract action relay	
	
	temperature		:REAL;// TMP Motor Temperature
	current			:REAL;// TMP Motor Current
	vol				:REAL;// TMP Voltage
	
	setpower		:UDINT;
	settime			:UDINT;

	enableOpen		: BOOL:=TRUE;//for outside control instance
	enableClose		: BOOL:=TRUE;//for outside control instance
	
	runTime			: LINT;
//state
	HMIEnable		: BOOL:=TRUE;
	enable			: BOOL;
	busy			: BOOL;
	done			: BOOL;
	error			: BOOL;
	Accerror		: BOOL;
	Dccerror		: BOOL;
	Alm				: BOOL;
	errID			: DINT;
	nameTXT			: STRING(255);//分子泵名称
	errTXT			: STRING;
	opencondition	: BOOL;// 开条件
	closecondition	: BOOL;// 关条件
END_STRUCT
END_TYPE
(*
按照字节对齐规则，将变量按字节大小按顺序定义，用于ADS读取
*)

// ---- POUs/BaseModule/ActionModule/TMPModule/enum/TMPType.TcDUT
TYPE TMPType :
(
	TMPType_Default := 0 //常规分子泵
)UINT;
END_TYPE

// ---- POUs/BaseModule/ActionModule/TMPModule/struct/TMPHMIStruts.TcDUT
{attribute 'pack_mode' := 1}
TYPE TMPHMIStruts :
STRUCT
	// Aiko
	singleControl: BOOL:=FALSE;//单控件触发信号
	singleControltemp: BOOL:=FALSE;//单控件触发信号
	bopen			: BOOL:=FALSE;//启动触发信号
	runTimeClear	: BOOL:=FALSE;//清空计时时间
//control signal or data
	open			: BOOL:=FALSE;//启动触发信号
	close			: BOOL:=FALSE;//停止触发信号
	reset			: BOOL:=FALSE;//复位信号
	stop			: BOOL:=FALSE;//停止信号
	power			: BOOL:=TRUE;//no power, two relay will lost power

//monitor
	AccAprSw		: BOOL:=FALSE;//HW: cylinder extent approach switch
	DccAprSw		: BOOL:=FALSE;//HW: cylinder retract approach switch	
	NormalAprSw		: BOOL:=FALSE;//HW: cylinder retract approach switch	
	AlmAprSw		: BOOL:=FALSE;//HW: cylinder retract approach switch
	ErrorAprSw		: BOOL:=FALSE;//HW: cylinder retract approach switch
	
	openRelay		: BOOL:=FALSE;//HW: cylinder extent action relay
	closeRelay		: BOOL:=FALSE;//HW: cylinder retract action relay	
	resetRelay		: BOOL:=FALSE;//HW: cylinder retract action relay	
	
	temperature		:REAL;// TMP Motor Temperature
	current			:REAL;// TMP Motor Current
	speed			:REAL;// TMP Motor MaxSpeed

	enableOpen		: BOOL:=TRUE;//for outside control instance
	enableClose		: BOOL:=TRUE;//for outside control instance
	
	runTime			: LINT;
//state
	HMIEnable		: BOOL:=TRUE;
	enable			: BOOL;
	busy			: BOOL;
	done			: BOOL;
	error			: BOOL;
	Accerror		: BOOL;
	Dccerror		: BOOL;
	Alm				: BOOL;
	errID			: DINT;
	nameTXT			: STRING(255);//分子泵名称
	errTXT			: STRING;
	opencondition	: BOOL;// 开条件
	closecondition	: BOOL;// 关条件
END_STRUCT
END_TYPE
(*
按照字节对齐规则，将变量按字节大小按顺序定义，用于ADS读取
*)

// ---- POUs/BaseModule/ActionModule/VPEModule/enum/VPEType.TcDUT
TYPE VPEType :
(
	VPEType_Default := 0 //常规泵组
)UINT;
END_TYPE

// ---- POUs/BaseModule/ActionModule/VPEModule/struct/VPEHMIStruts.TcDUT
{attribute 'pack_mode' := 1}
TYPE VPEHMIStruts :
STRUCT
//control signal or data
	extendAndretract: BOOL:=FALSE;//单控件触发信号
	runTimeClear	: BOOL:=FALSE;//清空计时时间
	singleControl				: BOOL:=FALSE;//单一信号控制
	singleControltemp			: BOOL:=FALSE;//单一信号控制
	open			: BOOL:=FALSE;//启动触发信号
	close			: BOOL:=FALSE;//停止触发信号
	reset			: BOOL:=FALSE;//复位信号
	stop			: BOOL:=FALSE;//停止信号
	power			: BOOL:=TRUE;//no power, two relay will lost power

//monitor
	
	openRelay		: BOOL:=FALSE;//HW: cylinder extent action relay
	
	DryPumpAlarm1	: UINT:=0;// 螺杆泵报警1
	DryPumpAlarm2	: UINT:=0;// 螺杆泵报警1
	DryPumpSpeed	: REAL:=0;// 螺杆泵速度
	DryPumpTemperature	: REAL:=0;// 螺杆泵温度
	DryPumpCurrent	: REAL:=0;// 螺杆泵电流
	DryPumpPower	: REAL:=0;// 螺杆泵功率
	DryPumpStart	: BOOL:=FALSE;// 螺杆泵启动
	DryPumpError	: BOOL:=FALSE;// 螺杆泵报错
	
	BoosterAlarm1	: UINT:=0;// 罗茨泵报警1
	BoosterAlarm2	: UINT:=0;// 罗茨泵报警1
	BoosterSpeed	: REAL:=0;// 罗茨泵速度
	BoosterTemperature	: REAL:=0;// 罗茨泵温度
	BoosterCurrent	: REAL:=0;// 罗茨泵电流
	BoosterPower	: REAL:=0;// 罗茨泵功率
	BoosterStart	: BOOL:=FALSE;// 罗茨泵启动
	BoosterError	: BOOL:=FALSE;// 罗茨泵报错
	
	Accing			: BOOL:=FALSE;// 泵组加速中
	Dccing			: BOOL:=FALSE;// 泵组减速中
	Normal			: BOOL:=FALSE;// 泵组全速中

	enableOpen		: BOOL:=TRUE;//for outside control instance
	enableClose		: BOOL:=TRUE;//for outside control instance
	
	runTime			: LINT;
	tailrowPre		: REAL;// 尾排压力
	AccAprSw		: BOOL;// 预热，加速
	AlmAprSw		: BOOL;// 报警
//state
	HMIEnable		: BOOL:=TRUE;
	enable			: BOOL;
	busy			: BOOL;
	done			: BOOL;
	error			: BOOL;
	errID			: DINT;
	nameTXT			: STRING;//泵组名称
	errTXT			: STRING;
	opencondition	: BOOL;// 开条件
	closecondition	: BOOL;// 关条件
END_STRUCT
END_TYPE
(*
按照字节对齐规则，将变量按字节大小按顺序定义，用于ADS读取
*)

// ---- POUs/BaseModule/ActionModule/VPEModule/struct/VPETestStruts530.TcDUT
{attribute 'pack_mode' := 1}
TYPE VPETestStruts530 :
STRUCT
	nouseData:DWORD;//报文头1 前4字节
	nouseData1:DWORD;//报文头2 后4字节
	nouseData4:BYTE;// 无用
	DryPumpState:DWORD;
	BoosteState:DWORD;
	FastStopState:DWORD;
	nouseData3:DWORD;// 无用
	DryPumpAlarm1:DWORD;
	BoosterAlarm1:DWORD;
	DryPumpAlarm2:DWORD;
	BoosterAlarm2:DWORD;
	DryPumpSpeed:DWORD;
	BoosterSpeed:DWORD;
END_STRUCT
END_TYPE
(*
按照字节对齐规则，将变量按字节大小按顺序定义，用于ADS读取
*)

// ---- POUs/BaseModule/ActionModule/VPEModule/struct/VPETestStruts540.TcDUT
{attribute 'pack_mode' := 1}
TYPE VPETestStruts540 :
STRUCT
	nouseData:DWORD;//报文头1 前4字节
	nouseData1:DWORD;//报文头2 后4字节
	nouseData4:BYTE;// 无用
	DryPumpTemp:DWORD;// 540
	nouseData2:DWORD;// 541
	BoosterTemp:DWORD;// 542
	nouseData3:DWORD;// 543
	DryPumpPower:DWORD;// 544
	BoosterPower:DWORD;// 545
	DryPumpCurrent:DWORD;// 546
	BoosterCurrent:DWORD;// 547
END_STRUCT
END_TYPE
(*
按照字节对齐规则，将变量按字节大小按顺序定义，用于ADS读取
*)

// ---- POUs/BaseModule/Communication/struct/struct_byte_1.TcDUT
TYPE struct_byte_1 :
STRUCT
	b1		:BYTE:=0;
	b2		:BYTE:=0;
	b3		:Byte:=0;
	b4		:Byte:=0;
	b5		:Byte:=0;
	b6		:Byte:=0;
	b7		:Byte:=0;
	b8		:Byte:=0;
	b9		:BYTE:=0;
	b10		:BYTE:=0;
	b11		:BYTE:=0;
	b12		:BYTE:=0;
	b13		:BYTE:=0;
	b14		:BYTE:=0;
	b15		:BYTE:=0;
	b16		:BYTE:=0;
	b17		:BYTE:=0;
	b18		:BYTE:=0;
	b19		:BYTE:=0;
	b20		:BYTE:=0;
END_STRUCT
END_TYPE

// ---- POUs/BaseModule/Communication/struct/struct_Tester.TcDUT
TYPE struct_Tester :
STRUCT
	channel		:DINT:=0;
	msgType		:DINT:=0;
	funCode		:DINT:=0;
	value1		:REAL:=0;
	value2		:REAL:=0;
	value3		:REAL:=0;
	value4		:REAL:=0;
	value5		:REAL:=0;
	errID		:LINT:=0;
	str			:STRING(g_nMaxByte_Client):='';
END_STRUCT
END_TYPE

// ---- POUs/BaseModule/Communication/struct/struct_byte.TcDUT
TYPE struct_byte :
STRUCT
	b1		:BYTE:=0;
	b2		:BYTE:=0;
	b3		:Byte:=0;
	b4		:Byte:=0;
	b5		:Byte:=0;
	b6		:Byte:=0;
	b7		:Byte:=0;
	b8		:Byte:=0;
	b9		:BYTE:=0;
	b10		:BYTE:=0;
	b11		:BYTE:=0;
	b12		:BYTE:=0;
	b13		:BYTE:=0;
	b14		:BYTE:=0;
	b15		:BYTE:=0;
	b16		:BYTE:=0;
	b17		:BYTE:=0;
	b18		:BYTE:=0;
	b19		:BYTE:=0;
	b20		:BYTE:=0;
END_STRUCT
END_TYPE

// ---- POUs/BaseModule/DataSaveModule_EX/Struct/RecipeNamePar.TcDUT
TYPE RecipeNamePar :
STRUCT
	NUM:STRING;
	Name:STRING;
	ID:STRING;
	Note1:STRING;
	Note2:STRING;
END_STRUCT
END_TYPE

// ---- POUs/BaseModule/DataSaveModule_EX/Struct/RecipePar.TcDUT
TYPE RecipePar :
STRUCT
	NUM:STRING;
	etchTime:STRING;
	rfPoint_Source:STRING;
	pdvPoint:STRING;
	mfc1:STRING;
	mfc2:STRING;
	mfc3:STRING;
	mfc4:STRING;
	mfc5:STRING;
	mfc6:STRING;
	mfc7:STRING;
	mfc8:STRING;
	mfc9:STRING;
	rfPoint_Power:STRING;
	par_2:STRING;
	par_3:STRING;
	par_4:STRING;
END_STRUCT
END_TYPE

// ---- POUs/BaseModule/DataSaveModule_EX/Struct/RecipeShowStr.TcDUT
TYPE RecipeShowStr :
STRUCT
	Name:STRING;
END_STRUCT
END_TYPE

// ---- POUs/BaseModule/EL2252_2262Control/struct/ST_CamSwitch.TcDUT
TYPE ST_CamSwitch :
STRUCT
	bTimeMode:BOOL:=TRUE;//TRUE表示时间控制模式, 持续时间由fDuration控制; FALSE表示位置控制模式，持续时间由fFirstOnPosition和fLastOnPosition控制
	fFirstOnPosition:LREAL;//时间控制模式和位置控制模式触发起始点
	fLastOnPosition:LREAL:=fFirstOnPosition+0.5;//位置控制模式触发结束点
	iAxisDirection:INT:=0;//-1表示负方向检测; 0表示正负方向检测(时间控制模式必须是0); 1表示正方向检测; 
	fDuration:LREAL:=5E-6;//持续时间, 单位s
END_STRUCT
END_TYPE

// ---- POUs/BaseModule/EL2252_2262Control/struct/ST_CamSwitch_EL2262.TcDUT
TYPE ST_CamSwitch_EL2262 :
STRUCT
	bTimeMode:BOOL:=TRUE;//TRUE表示时间控制模式, 持续时间由fDuration控制; FALSE表示位置控制模式，持续时间由fFirstOnPosition和fLastOnPosition控制
	fFirstOnPosition:LREAL;//时间控制模式和位置控制模式触发起始点
	fLastOnPosition:LREAL:=fFirstOnPosition+0.5;//位置控制模式触发结束点
	iAxisDirection:INT:=0;//-1表示负方向检测; 0表示正负方向检测(时间控制模式必须是0); 1表示正方向检测;
	fDuration:LREAL:=5E-6;//持续时间, 单位s
END_STRUCT
END_TYPE

// ---- POUs/BaseModule/EL2252_2262Control/struct/ST_EL2262OutData.TcDUT
TYPE ST_EL2262OutData :
STRUCT
	Output0 					AT%Q*:ARRAY[0..124] OF BYTE;
	Output1 					AT%Q*:ARRAY[0..124] OF BYTE;
END_STRUCT
END_TYPE

// ---- POUs/BaseModule/Error/enum/Error_Level.TcDUT
//{attribute 'qualified_only'}
//{attribute 'strict'}
TYPE Error_Level ://报错等级 
(
	//Error_Level_Def		:= -1,//不上报ALC，仅在PLC打印显示
	Error_Level_0		:= 0,//报错等级 0 设备不暂停，ALC仅仅做记录，不提示
	Error_Level_1		:= 1,//报错等级 1 设备不暂停，ALC仅仅做记录，不提示
	Error_Level_2		:= 2,//报错等级 2 设备不暂停，ALC弹框提示，不会触发PLC做任何处理
	Error_Level_3		:= 3,//报错等级 3 设备暂停，ALC弹框提示，可以选择继续或停机
	Error_Level_4		:= 4 //报错等级 4 设备退出运行，ALC弹框提示
)INT;
END_TYPE

// ---- POUs/BaseModule/Error/struct/ST_Error.TcDUT
TYPE ST_Error :
STRUCT
	bError				:BOOL;
	uErrID				:LINT;//Error ID
	sErrTXT				:STRING(255);//Error TXT //g_nMaxByte_Client
	sErrWTXT			:WSTRING(255);//Error TXT //g_nMaxByte_Client
	eErrLevel			:Error_Level:=Error_Level.Error_Level_3;//Error Level
END_STRUCT
END_TYPE

// ---- POUs/BaseModule/IO/ReadWriteCSV/ST_DataFmtBase.TcDUT
TYPE ST_DataFmtBase :
STRUCT
	nGroup:DINT;
	nNumber:DINT;
	sTxt_ENG:STRING;
	sTxt_CHN:WSTRING;
END_STRUCT
END_TYPE

// ---- POUs/BaseModule/IO/struct/ST_INPUT_IO.TcDUT
TYPE ST_INPUT_IO :
STRUCT
	io AT%I*:ARRAY [1..16] OF BOOL;
END_STRUCT
END_TYPE

// ---- POUs/BaseModule/IO/struct/ST_IOBase_Show_HMI.TcDUT
{attribute 'pack mode' := 1}
TYPE ST_IOBase_Show_HMI :
STRUCT
	bIO:ARRAY [1..16] OF BOOL;
	iInfor:ARRAY [1..16] OF DINT;
	sInfor:ARRAY [1..16] OF WSTRING;
	iMaxPage:DINT:=1;
	iCurrPage:DINT:=1;
	iTargerPage:DINT:=1;
	bNextPage:BOOL;
	bBackPage:BOOL;
	bTargerPage:BOOL;
	sIOType:STRING:='Input';// 'Input' or 'Output'
END_STRUCT
END_TYPE

// ---- POUs/BaseModule/IO/struct/ST_OUTPUT_IO.TcDUT
TYPE ST_OUTPUT_IO :
STRUCT
	io AT%Q*:ARRAY [1..16] OF BOOL;
END_STRUCT
END_TYPE

// ---- POUs/BaseModule/MainFrame/MainFram.TcDUT
TYPE MainFram :
STRUCT
	ComName			:STRING:='CYG_Vision';//公司名称
	ProjectName		:STRING:='Marimba';//项目名称	
	ShowTime		:STRING:='';//当前时间显示变量
	
	StartLamp		:BOOL;//启面急停动指示
	ResetLamp		:BOOL;//复面急停位指示
	StopLamp		:BOOL;//停面急停止，报错指示
	
	E_Stop			:BOOL:=TRUE;//界面急停显示
	Start			:BOOL;//界面启动
	Reset			:BOOL;//界面复位
	Stop			:BOOL;//界面停止
	
	GreenLamp		:BOOL;//界面启动按钮灯
	YellowLamp		:BOOL;//界面复位动按钮灯
	RedLamp			:BOOL;//界面停止动按钮灯
	
	Loading			:BOOL;//界面登录
	Quit			:BOOL;//界面退出
	versions		:STRING;//版本号
	RunStateTxt		:WSTRING;//运行状态
	ErrWTxtShow		:WSTRING;//错误状态
	CtrlMode		:ControlMode;//控制模式
	
END_STRUCT
END_TYPE

// ---- POUs/BaseModule/PrintLogModule_EX/struct/printLogModule_EX_DataHMI.TcDUT
{attribute 'pack mode' := 1}
TYPE printLogModule_EX_DataHMI :
STRUCT
	logStrData			:ARRAY [cNumBegin_showInof..cNumLength_showInof] OF printLogModule_EX_DataST;
	enableSave			:BOOL:=FALSE;
	enableSaveShowLog	:BOOL:=FALSE;
	clearInformation	:BOOL:=FALSE;
END_STRUCT
END_TYPE

// ---- POUs/BaseModule/PrintLogModule_EX/struct/printLogModule_EX_DataST.TcDUT
TYPE printLogModule_EX_DataST :
STRUCT
	sTime			:WSTRING(255);
	msg				:WSTRING(255);//T_MaxString
END_STRUCT
END_TYPE

// ---- POUs/BaseModule/PrintLogModule_EX/struct/ST_DeleteFile.TcDUT
TYPE ST_DeleteFile :
STRUCT
	sDirPath:STRING;//目录路径名
	sFilePath:STRING;//文件路径名
	nCount:UINT;//计数
END_STRUCT
END_TYPE

// ---- POUs/BaseModule/TcpIpModule_EX/dataStruct_EX/ST_TCPIP_DATA_STRUCT_ALC.TcDUT
TYPE ST_TCPIP_DATA_STRUCT_ALC :
STRUCT
	channel		:DINT;
	msgType		:DINT;
	funCode		:DINT;
	value1		:REAL;
	value2		:REAL;
	value3		:REAL;
	value4		:REAL;
	value5		:REAL;
	errID		:LINT;
	str			:ARRAY[1..g_nMaxByte_Client] OF BYTE;
END_STRUCT
END_TYPE
(*
结构体的数据结构需要按照与上位机制定的格式设定
*)

// ---- POUs/Communication/Communica_ALC/enum_CommandNumber.TcDUT
{attribute 'qualified_only'}
{attribute 'strict'}
TYPE enum_CommandNumber :
(
	enum_member := 0
)DINT;
END_TYPE

// ---- POUs/Communication/Communica_ALC/E_Sta1_CMD.TcDUT
{attribute 'qualified_only'}
{attribute 'strict'}
TYPE E_Sta1_CMD :
(
	enum_resign:=1,//注册
	enum_Init:=2,//初始化

	enum_test_start := 3,	// 启动
	enum_test_stop := 4,	// 停止
	enum_test_reset := 5,	// 复位
	enum_test_pause := 6,	// 暂停
	enum_test_resume :=7,	// 恢复
	
	enum_DUTchange := 8,	// 产品检测类型切换：MsgType=0尺寸   MsgType=1缺陷
	enum_sizechange := 9,	// 产品尺寸切换：MsgType=0大尺寸  MsgType=1小尺寸
	enum_modechange := 10,	// 模式切换：MsgType=0离线   MsgType=1在线
	
	enum_test_error := 99,	// 报错
	
	enum_SWsensingmaterial := 130,	// 主控：感应到物料
	enum_SWrequestdownload := 140,	// 主控：请求下料
	enum_SWrequestdownload_twince := 141,	// 主控：二次请求分BIN
	enum_SWCMD_Stop := 201,	// 软件要求停机
	enum_SWCMD_UnloadAOI1 := 555,	// AOI1-PhotoTOUnloadDUT
	enum_SWCMD_GrrInit:=700,
	enum_SWCMD_GrrReady:=600,
	
//	enum_Photo1 := 21,// Photo1
//	enum_Photo2 := 41,// Photo2
//	enum_Photo3 := 51,// Photo3
//	enum_Photo4 := 61,// Photo4
//	enum_Photo5 := 71,// Photo5
//	enum_Photo6 := 81,// Photo6
//	enum_Photo7 := 91,// Photo7
//	enum_Photo8 := 101,// Photo8
//	enum_Photo9 := 111,// Photo9
//	enum_Photo10 := 121,// Photo10
//	enum_Photo11 := 131,// Photo11
//	enum_Photo12 := 31,// Photo12
	
//	enum_Photo13 := 31,	// Photo13
//	enum_Photo14 := 31,	// Photo14
//	enum_Photo15 := 31	// Photo15

//编排顺序对应软件的STA1-STA12，从301开始到312接收，因12相机处于STA1和STA2之间，因此无法对应工站号
	enum_Photo1 := 301,// Photo1
	enum_Photo2 := 302,// Photo2
	enum_Photo3 := 303,// Photo3
	enum_Photo4 := 304,// Photo4
	enum_Photo5 := 305,// Photo5
	enum_Photo6 := 306,// Photo6
	enum_Photo7 := 307,// Photo7
	enum_Photo8 := 308,// Photo8
	enum_Photo9 := 309,// Photo9
	enum_Photo10 := 310,// Photo10
	enum_Photo11 := 311,// Photo11
	enum_Photo12 := 312,// Photo12
	enum_Photo13 := 313,// Photo13
	enum_Photo14 := 314,// Photo14
	enum_Photo15 := 315	 // Photo15

	
);
END_TYPE

// ---- POUs/Other/ActBase/ITF/struct/ST_ActStep_State.TcDUT
TYPE ST_ActStep_State :
STRUCT
	step:DINT;//当前运行的step
	errStep:DINT;//跳转到error状态的step
	nextStep:DINT;//paused解除之后的下一步step
	
	ex:BOOL;//执行触发
	pause:BOOL;//暂停触发，效果：不跳转到下一步
	paused:BOOL;//paused 状态
	
	busy:BOOL;//busy 状态
	done:BOOL;//done 状态
	error:BOOL;//error 状态
	errID:DINT;//error ID
	errMsg:STRING(255);//error 信息
END_STRUCT
END_TYPE

// ---- POUs/Other/HMI/WARMStruct.TcDUT
TYPE WARMStruct :
STRUCT
	showText		:STRING:='********';// 提示内容
	showFlag		:BOOL;// 提示显示
	btTrig			:BOOL;// 触发按钮			
	bOK				:BOOL;
	bNO				:BOOL;
END_STRUCT
END_TYPE

// ---- POUs/Other/HMI/NoteStruct.TcDUT
TYPE NoteStruct :
STRUCT
	showText		:STRING:='********';// 提示内容
	showFlag		:BOOL;// 提示显示			
	bOK				:BOOL;
	bNO				:BOOL;
END_STRUCT
END_TYPE

// ---- POUs/Other/MachineState/enum/RunningStatus.TcDUT
TYPE RunningStatus :
(
	eManualState	:= 1,//手动状态
	eAutoState	 	:= 2,//自动状态
	ePauseState		:= 3,//暂停状态
	eStopState		:= 4,//停止状态
	eErrorState		:= 5,//错误状态
	eHomeState		:= 6 //回原点状态
)UINT;
END_TYPE

// ---- POUs/Other/MachineState/ST_DownTimeRecord.TcDUT
TYPE ST_DownTimeRecord :
STRUCT
	startTime:TIME;
	endTime:TIME;
	start2end_time:TIME;
	start2end_ms:UDINT;// 开始到结束的总时间，ms单位
	start2end_s:LREAL;// 开始到结束的总时间，s单位
	record_s:LREAL;// 时间记录，s单位
	
	bMonitor:BOOL;// 监控条件
	
	rTrig:R_TRIG;
	fTrig:F_TRIG;
END_STRUCT
END_TYPE

// ---- POUs/Other/MachineState/ST_MachineState.TcDUT
TYPE ST_MachineState :
STRUCT
	HMI_E_Stop				:BOOL:=TRUE;
	HMI_Start				:BOOL:=FALSE;
	HMI_Stop				:BOOL:=FALSE;
	HMI_Reset				:BOOL:=FALSE;
	HMI_EnableBuzzer		:BOOL:=FALSE;
	HMI_RunStateTxt			:STRING:='';
	Actual_E_Stop			:BOOL;//设备 EStop 按钮-
	Actual_Start			:BOOL;//设备 Start 按钮
	Actual_Stop				:BOOL;//设备 Stop 按钮
	Actual_Reset			:BOOL;//设备 Reset 按钮
	Actual_StartLamp		:BOOL;//设备 Start 按钮灯
	Actual_StopALamp		:BOOL;//设备 Stop 按钮灯
	Actual_ResetLamp		:BOOL;//设备 Reset 按钮灯
	Actual_RedLamp			:BOOL;//设备 三色灯 Red 灯
	Actual_YellowLamp		:BOOL;//设备 三色灯 Yellow 灯
	Actual_GreenLamp		:BOOL;//设备 三色灯 Green 灯
	Actual_Buzzer			:BOOL;//设备 三色灯 Buzzer
END_STRUCT
END_TYPE

// ---- POUs/Other/Struct/ActPos/ST_DOEActPos.TcDUT
TYPE ST_DOEActPos :
STRUCT
	X1LoadPos:LREAL;//Tray盘上料位，靠近确认按钮侧
	X1SafePos:LREAL;//Tray盘移动安全位
	X1UnLoadPos:LREAL;//Tray下料位，即吸嘴上料位
	X1ScanPos:LREAL;//X1扫码位
	
	Y1LoadPos:LREAL;//吸嘴Y1模组上料位
	Y1PhotoPos:LREAL;//上料上相机拍照位(Y1移动)
	Y1SafePos:LREAL;//上料Y1模组安全位
	Y1UnLoadPos:LREAL;//上料Y1模组下料至载具安全位
	Y1NGUnLoadPos:LREAL;//Y1轴NG下料位置
	Y1ScanPos:LREAL;// Y1扫码位
	Y1LoadPhotoPos:LREAL;//载具下料——上料拍照位
	
	Z1LoadPos:LREAL;//上料吸嘴Z1上料高度
	Z1LoadSafePos:LREAL;//上料吸嘴Z1轴上料安全高度
	Z1SafePos:LREAL;//上料吸嘴Z1轴在Y1轴移动时的安全高度
	Z1UnLoadSafePos:LREAL;//上料吸嘴Z1轴下料安全高度
	Z1UnLoadPos:LREAL;//上料吸嘴Z1轴下料至载具高度
	Z1NGUnLoadPos:LREAL;//Z1轴NG下料位置
	
	
	R1InitPos:LREAL;//上料吸嘴R1轴初始角度（手动对位值）
	R1LoadPos:LREAL;//上料吸嘴取料角度
	R1TopBottomPos:LREAL;//上料吸嘴R1拍姿态角度
	R1UnLoadPos:LREAL;//上料吸嘴下料角度
	
	CY1SafePos:LREAL;//上料相机CY1安全位（避让Socket移动）
	CY1PhotoPos:LREAL;//上料相机景深工作位CY1:有可能只要工作位
	CY1TopPhotoPos:LREAL;//载具GRR拍物料Top圆
	
	
END_STRUCT
END_TYPE

// ---- POUs/Other/Struct/StationBuild/ST_ICP.TcDUT
TYPE ST_ICP :
STRUCT
	// 干泵
	MachianicalPum								:VPEModule;
	MachianicalPumAcc							:BOOL;//预热，加速信号
	MachianicalPumAlm							:BOOL;//泵组报警信号
	MachianicalPumOpen							:BOOL;//泵组开继电器
	// 阀门
	// 1
	ForlinLineValve								:CylinderModule;
	ForlinLineValveExtRelay						:BOOL;// 输出变量,开阀线圈
	ForlinLineValveNoteArry						:ARRAY [1..gNoteArryMaxNum] OF WSTRING;// 操作提示
	// 2
	RoughValve									:CylinderModule;
	RoughValveExtRelay							:BOOL;// 输出变量,开阀线圈
	RoughValveNoteArry							:ARRAY [1..gNoteArryMaxNum] OF WSTRING;// 操作提示
	// 3
	SlowPummingValve							:CylinderModule;
	SlowPummingExtRelay							:BOOL;// 输出变量,开阀线圈
	SlowPummingNoteArry							:ARRAY [1..gNoteArryMaxNum] OF WSTRING;// 操作提示
	// 4
	FastPummingValve							:CylinderModule;
	FastPummingExtRelay							:BOOL;// 输出变量,开阀线圈
	FastPummingNoteArry							:ARRAY [1..gNoteArryMaxNum] OF WSTRING;// 操作提示
	// 5
	ElectrodeCyl								:CylinderModule;
	ElectrodeCylExtRelay						:BOOL;// 输出变量,开阀线圈
	ElectrodeCylRetRelay						:BOOL;// 输出变量,关阀线圈
	ElectrodeCylExtSensor						:BOOL;// 输入变量,开到位
	ElectrodeCylRetSensor						:BOOL;// 输入变量,关到位
	ElectrodeCylNoteArry						:ARRAY [1..gNoteArryMaxNum] OF WSTRING;// 操作提示
	// 6
	LiftPinCyl									:CylinderModule;
	LiftPinExtRelay								:BOOL;// 输出变量,开阀线圈
	LiftPinRetRelay								:BOOL;// 输出变量,关阀线圈
	LiftPinExtSensor							:BOOL;// 输入变量,开到位
	LiftPinRetSensor							:BOOL;// 输入变量,关到位
	LiftPinNoteArry								:ARRAY [1..gNoteArryMaxNum] OF WSTRING;// 操作提示
	// 7
	GVA1Valve									:CylinderModule;
	GVA1ExtRelay								:BOOL;// 输出变量,开阀线圈
	GVA1NoteArry								:ARRAY [1..gNoteArryMaxNum] OF WSTRING;// 操作提示
	// 8
	GVA2Valve									:CylinderModule;
	GVA2ExtRelay								:BOOL;// 输出变量,开阀线圈
	GVA2NoteArry								:ARRAY [1..gNoteArryMaxNum] OF WSTRING;// 操作提示
	// 9
	GVA3Valve									:CylinderModule;
	GVA3ExtRelay								:BOOL;// 输出变量,开阀线圈
	GVA3NoteArry								:ARRAY [1..gNoteArryMaxNum] OF WSTRING;// 操作提示
	// 10
	GVA4Valve									:CylinderModule;
	GVA4ExtRelay								:BOOL;// 输出变量,开阀线圈
	GVA4NoteArry								:ARRAY [1..gNoteArryMaxNum] OF WSTRING;// 操作提示
	// 11
	GVA5Valve									:CylinderModule;
	GVA5ExtRelay								:BOOL;// 输出变量,开阀线圈
	GVA5NoteArry								:ARRAY [1..gNoteArryMaxNum] OF WSTRING;// 操作提示
	// 12
	GVA6Valve									:CylinderModule;
	GVA6ExtRelay								:BOOL;// 输出变量,开阀线圈
	GVA6NoteArry								:ARRAY [1..gNoteArryMaxNum] OF WSTRING;// 操作提示
	// 13
	GVA7Valve									:CylinderModule;
	GVA7ExtRelay								:BOOL;// 输出变量,开阀线圈
	GVA7NoteArry								:ARRAY [1..gNoteArryMaxNum] OF WSTRING;// 操作提示
	// 14
	GVA8Valve									:CylinderModule;
	GVA8ExtRelay								:BOOL;// 输出变量,开阀线圈
	GVA8NoteArry								:ARRAY [1..gNoteArryMaxNum] OF WSTRING;// 操作提示
	// 15
	GVA9Valve									:CylinderModule;
	GVA9ExtRelay								:BOOL;// 输出变量,开阀线圈
	GVA9NoteArry								:ARRAY [1..gNoteArryMaxNum] OF WSTRING;// 操作提示
	// 16
	GVA10Valve_Vent								:CylinderModule;
	GVA10ExtRelay_Vent							:BOOL;// 输出变量,开阀线圈--Vent  N2
	GVA10NoteArry_Vent							:ARRAY [1..gNoteArryMaxNum] OF WSTRING;// 操作提示
	
	// 16
	GV20Valve_Main								:CylinderModule;
	GV20ExtRelay_Main							:BOOL;// 输出变量,开阀线圈--MainValve
	GV20NoteArry_Main							:ARRAY [1..gNoteArryMaxNum] OF WSTRING;// 操作提示
	
	// 17
	GVB1Valve									:CylinderModule;
	GVB1ExtRelay								:BOOL;// 输出变量,开阀线圈
	GVB1NoteArry								:ARRAY [1..gNoteArryMaxNum] OF WSTRING;// 操作提示
	// 18
	GVB2Valve									:CylinderModule;
	GVB2ExtRelay								:BOOL;// 输出变量,开阀线圈
	GVB2NoteArry								:ARRAY [1..gNoteArryMaxNum] OF WSTRING;// 操作提示
	// 19
	GVB3Valve									:CylinderModule;
	GVB3ExtRelay								:BOOL;// 输出变量,开阀线圈
	GVB3NoteArry								:ARRAY [1..gNoteArryMaxNum] OF WSTRING;// 操作提示
	// 20
	GVB4Valve									:CylinderModule;
	GVB4ExtRelay								:BOOL;// 输出变量,开阀线圈
	GVB4NoteArry								:ARRAY [1..gNoteArryMaxNum] OF WSTRING;// 操作提示
	// 21
	GVB5Valve									:CylinderModule;
	GVB5ExtRelay								:BOOL;// 输出变量,开阀线圈
	GVB5NoteArry								:ARRAY [1..gNoteArryMaxNum] OF WSTRING;// 操作提示
	// 22
	GVB6Valve									:CylinderModule;
	GVB6ExtRelay								:BOOL;// 输出变量,开阀线圈
	GVB6NoteArry								:ARRAY [1..gNoteArryMaxNum] OF WSTRING;// 操作提示
	// 23
	GVB7Valve									:CylinderModule;
	GVB7ExtRelay								:BOOL;// 输出变量,开阀线圈
	GVB7NoteArry								:ARRAY [1..gNoteArryMaxNum] OF WSTRING;// 操作提示
	// 24
	GVB8Valve									:CylinderModule;
	GVB8ExtRelay								:BOOL;// 输出变量,开阀线圈
	GVB8NoteArry								:ARRAY [1..gNoteArryMaxNum] OF WSTRING;// 操作提示
	// 25
	GVB9Valve									:CylinderModule;
	GVB9ExtRelay								:BOOL;// 输出变量,开阀线圈
	GVB9NoteArry								:ARRAY [1..gNoteArryMaxNum] OF WSTRING;// 操作提示
	// 26
	ISOValve								     :CylinderModule;
	ISOExtRelay								     :BOOL;// 输出变量,开阀线圈
	ISONoteArry								     :ARRAY [1..gNoteArryMaxNum] OF WSTRING;// 操作提示
	
	// 27
	AIMValve								     :CylinderModule;
	AIMExtRelay								     :BOOL;// 输出变量,开阀线圈
	AIMNoteArry								     :ARRAY [1..gNoteArryMaxNum] OF WSTRING;// 操作提示
	
	//28
	GateDoorValve								 :CylinderModule;
	GateDoorExtRelay							 :BOOL;// 输出变量,开阀线圈
	GateDoorRetRelay							 :BOOL;// 输出变量,关阀线圈
	GateDoorExtSensor							 :BOOL;// 输入变量,开到位
	GateDoorRetSensor							 :BOOL;// 输入变量,关到位
	GateDoorNoteArry							 :ARRAY [1..gNoteArryMaxNum] OF WSTRING;// 操作提示
	
	//29
	VentValve									 :CylinderModule;
	VentExtRelay								 :BOOL;// 输出变量,开阀线圈
	VentNoteArry								 :ARRAY [1..gNoteArryMaxNum] OF WSTRING;// 操作提示
	// 分子泵
	TruboPum									 :TMPModule;
	TruboPumAcc									 :BOOL;// 分子泵加速IO输入
	TruboPumNormal								 :BOOL;// 分子泵匀速IO输入
	TruboPumDcc									 :BOOL;// 分子泵减速IO输入
	TruboPumError								 :BOOL;// 分子泵报错IO输入
	TruboPumOpen								 :BOOL;// 分子泵启动IO输出
	TruboPumReset								 :BOOL;// 分子泵复位IO输出
	TruboPumNoRotation							 :BOOL; // 静止
	TruboPumAlarm								 :BOOL;	// 警告
	TruboPumRemote								 :BOOL;	// 远程操作中 远程操作为1
	TruboPumRotationSpeed						 :UDINT;// 实时转速（HZ）
	TruboPumTMS									 :REAL;// TMS 温度
	TruboPumNoteArry							 :ARRAY [1..gNoteArryMaxNum] OF WSTRING;// 操作提示
	
	// MFC
	MFC1										 :MFCModule;
	MFC1NoteArry								 :ARRAY [1..gNoteArryMaxNum] OF WSTRING;// 操作提示
	
	MFC2										 :MFCModule;
	MFC2NoteArry								 :ARRAY [1..gNoteArryMaxNum] OF WSTRING;// 操作提示
	
	MFC3										 :MFCModule;
	MFC3NoteArry								 :ARRAY [1..gNoteArryMaxNum] OF WSTRING;// 操作提示
	
	MFC4										 :MFCModule;
	MFC4NoteArry								 :ARRAY [1..gNoteArryMaxNum] OF WSTRING;// 操作提示
	
	MFC5										 :MFCModule;
	MFC5NoteArry								 :ARRAY [1..gNoteArryMaxNum] OF WSTRING;// 操作提示
	
	MFC6										:MFCModule;
	MFC6NoteArry								:ARRAY [1..gNoteArryMaxNum] OF WSTRING;// 操作提示
	
	MFC7										:MFCModule;
	MFC7NoteArry								:ARRAY [1..gNoteArryMaxNum] OF WSTRING;// 操作提示
	
	MFC8										:MFCModule;
	MFC8NoteArry								:ARRAY [1..gNoteArryMaxNum] OF WSTRING;// 操作提示
	
	MFC9										:MFCModule;
	MFC9NoteArry								:ARRAY [1..gNoteArryMaxNum] OF WSTRING;// 操作提示
	
	// RF 电源
	PowerRF										:RFModule;
	PowerRFOpenRelay							:BOOL;
	PowerRFResetRelay							:BOOL;
	PowerRF_Alrm								:BOOL;
	PowerRF_ON									:BOOL;
	PowerRFNoteArry								:ARRAY [1..gNoteArryMaxNum] OF WSTRING;// 操作提示
	
	SourceRF									:RFModule_Source;
	SourceRFOpenRelay							:BOOL;
	SourceRFResetRelay							:BOOL;
	SourceRF_Alrm								:BOOL;
	SourceRF_ON									:BOOL;
	SourceRFNoteArry							:ARRAY [1..gNoteArryMaxNum] OF WSTRING;// 操作提示
	
	// Chiller
	Chiller										:ChillerModule_1;// 水冷
	
	// PendulumValve
	PDV											:PVModule;
	PDVOpenRelay								:BOOL;// 输出变量,开阀线圈
	PDVCloseRelay								:BOOL;// 输出变量,关阀线圈
	PDVModeRelay								:BOOL;// 输出变量,模式切换线圈
	PDVOpenSensor								:BOOL;// 输入变量,开到位
	PDVCloseSensor								:BOOL;// 输入变量,关到位
	PDVNoteArry									:ARRAY [1..gNoteArryMaxNum] OF WSTRING;// 操作提示
	
	// ARM
	ARM											:ARMModule;
	I_ARMHome									:BOOL;
	// ATM
	I_ATMSensor									:BOOL;		
	
	// ForeLineGauge
	ForeLineGauge								:GaugeViewModule;
	AI_ForeLineGauge							AT %I* :INT ;
	// AIMGauge
	AIMGauge									:GaugeViewModule;
	AI_AIMGauge									AT %I* :INT ;
	// LoadLockGauge
	LoadLockGauge								:GaugeViewModule;
	AI_LoadLockGauge							AT %I* :INT ;
	// ChamberGauge
	ChamberGauge								:ChamberGaugeViewModule;
	AI_ChamberGauge								AT %I* :INT ;
	ChamberGaugeReal							:REAL;
	// TBGauge
	TBGauge										:GaugeViewModule;
	AI_TBGauge									:UDINT ;
	// HeMFM
	HeMFC_ActFlow								AT %I* :REAL ;
	HeMFC_SetFlow								AT %Q* :REAL:=2.5 ;
	HeMFC_SetFlowHMI							:REAL:=2 ;
	//30
	HeINValve									 :CylinderModule;
	HeINExtRelay								 :BOOL;// 输出变量,开阀线圈
	HeINNoteArry								 :ARRAY [1..gNoteArryMaxNum] OF WSTRING;// 操作提示
	//31
	HePumValve									 :CylinderModule;
	HePumExtRelay								 :BOOL;// 输出变量,开阀线圈
	HePumNoteArry								 :ARRAY [1..gNoteArryMaxNum] OF WSTRING;// 操作提示
	//32
	GASBoxVentValve								 :CylinderModule;
	GASBoxVentExtRelay							 :BOOL;// 输出变量,开阀线圈
	GASBoxVentNoteArry							 :ARRAY [1..gNoteArryMaxNum] OF WSTRING;// 操作提示
	
	//33
	TBPurgeValve								 :CylinderModule;
	TBPurgeExtRelay								 :BOOL;// 输出变量,开阀线圈
	TBPurgeNoteArry								 :ARRAY [1..gNoteArryMaxNum] OF WSTRING;// 操作提示
	// IO
	I_LLSwitch									:BOOL;// Load Lock Switch
	I_LLSwitchString							:STRING;
	I_WaferCheck								:BOOL;// Load Loch WaferCheck
	I_PressureCheck								:BOOL;// Pressure detection
	I_WaterFlowCheck							:BOOL;// WaterFlow detection
	I_WaterTemperatureCheck						:BOOL;// WaterTemperature detection
	I_ArmHomeSensor								:BOOL;// ARM Homeing Sensor
	HeCheckGaugeReal							:REAL;
	
	C_GASBOX_AllGVAOpen							:BOOL;// 全部GVAOpen
	C_GASBOX_AllGVBOpen							:BOOL;// 全部GVBOpen
	C_GASBOX_AllGVAClose						:BOOL;// 全部GVAClose
	C_GASBOX_AllGVBClose						:BOOL;// 全部GVBClose
	
	C_GASBOX_AllGVAOpenTemp						:BOOL;// 全部GVAOpen HMI
	C_GASBOX_AllGVBOpenTemp						:BOOL;// 全部GVBOpen HMI
	C_GASBOX_AllGVACloseTemp					:BOOL;// 全部GVAClose HMI
	C_GASBOX_AllGVBCloseTemp					:BOOL;// 全部GVBClose HMI
	
	C_GASBOX_AllGVOpen							:BOOL;// 全部GVOpen 
	C_GASBOX_AllGVClose							:BOOL;// 全部GVClose
	
	C_GASBOX_AllMFCSet							:BOOL;// 全部MFC设置
	C_GASBOX_AllMFCClear						:BOOL;// 全部MFC清除
	C_GASBOX_AllMFCSetTemp						:BOOL;// 全部MFC设置
	C_GASBOX_AllMFCClearTemp					:BOOL;// 全部MFC清除
	
	S_GASBOX_AllGVAOpen							:BOOL;// 全部GVAOpen 完成
	S_GASBOX_AllGVBOpen							:BOOL;// 全部GVBOpen 完成
	S_GASBOX_AllGVAClose						:BOOL;// 全部GVAClose 完成
	S_GASBOX_AllGVBClose						:BOOL;// 全部GVBClose 完成
	S_GASBOX_AllGVOpen							:BOOL;// 全部GVOpen 完成
	S_GASBOX_AllGVClose							:BOOL;// 全部GVClose 完成
	S_GASBOX_AllMFCSetDone						:BOOL;// 全部MFC设置 完成
	S_GASBOX_AllMFCClearDone					:BOOL;// 全部MFC清除 完成
	S_GASBOX_AllMFCClearDoneStep				:BOOL;// 全部MFC清除 完成
	S_GASBOX_AllMFCSetEqual						:BOOL;// 全部MFC设置参数 等于 反馈参数
	
	S_MFCMonitFlowNotZero						:BOOL;// MFC实时检查参数不小于0
END_STRUCT
END_TYPE

// ---- POUs/Other/Struct/ST_HaveDUTState.TcDUT
TYPE ST_HaveDUTState :
STRUCT
	haveDUT:BOOL;
	DutCheckDone:BOOL;
	DutCheckRuslut:BOOL;
END_STRUCT
END_TYPE

// ---- POUs/Other/Struct/ST_MachineUtility.TcDUT
TYPE ST_MachineUtility :
STRUCT
  	(*外罩按钮及三色灯*)
 	I_Start:BOOL;// 测试机 Start 按钮
	I_Stop:BOOL;// 测试机 Stop 按钮
	I_Reset:BOOL;// 测试机 Reset 按钮
	I_EStop:BOOL;// 测试机 E-Stop 按钮
	
 	O_StartLamp:BOOL;// 测试机 Start 按钮
	O_StopLamp:BOOL;// 测试机 Stop 按钮
	O_ResetLamp:BOOL;// 测试机 Reset 按钮
	O_RedLamp:BOOL;// 测试机 三色灯 红灯
	O_GreenLamp:BOOL;// 测试机 三色灯 绿灯
	O_YellowLamp:BOOL;// 测试机 三色灯 黄灯
	O_Buzzer:BOOL;// 测试机 三色灯 蜂鸣器
	
 	(*安全门信号*)
 	I_SafeDoor_1:BOOL;// 前安全门1
	I_SafeDoor_2:BOOL;// 后安全门1
	I_SafeDoor_3:BOOL;// 前安全门2
	I_SafeDoor_4:BOOL;// 后安全门2

	(*压力检测*)
	I_PressureDetection1:BOOL;
	(* 温度检测*)
	I_Temperature:BOOL;
END_STRUCT
END_TYPE

// ---- POUs/Other/Struct/ST_POUCommunication.TcDUT
TYPE ST_POUCommunication :
STRUCT
	CanLoad:BOOL;//允许上料
	LoadDone:BOOL;//上料完成
	
	SafePosConfirm:BOOL;//安全位置确认
	SafePosConfirmUnLoad:BOOL;//下料安全位置确认
	
	LoadCanHandle:BOOL;//允许交接,上料
	LoadHandleDone:BOOL;//交接完成,上料
	
	CanUnLoad:BOOL;//允许下料
	UnLoadDone:BOOL;//下料完成
	
	UnLoadCanHandle:BOOL;//允许交接,上料
	UnLoadHandleDone:BOOL;//交接完成,上料
	
	cantoUnload:BOOL;//允许测试载具直接到下料位
END_STRUCT
END_TYPE

// ---- POUs/Other/Struct/ST_StationConfigBase.TcDUT
TYPE ST_StationConfigBase :
STRUCT
	Pos1						:LREAL;//大尺寸物料——相机聚焦位置
	Move_Pos1					:BOOL;//移动到大尺寸物料相机聚焦位
	SavePar						:BOOL;//参数保存
	AixActVel					:LREAL;//轴对象实际速度
	AixActPos					:LREAL;//轴对象实际位置
	AixNameShow					:WSTRING;//现实名称
	AixChineseName				:WSTRING;//中文名称
	AixEnglishName				:STRING;//英文名称
	RunVel						:LREAL;//运行速度
	Stop						:BOOL;//运动复位
	Reset						:BOOL;//运动停止
	moveerror					:BOOL;//运动出错
	pos1name					:WSTRING:="位置1";
	savepos1btname				:WSTRING:="保存位置1";
	movetopos1btname			:WSTRING:="移动到位置1";
END_STRUCT
END_TYPE

// ---- GVLs/GVL_AllCONSTANT.TcGVL
//{attribute 'qualified_only'}
VAR_GLOBAL CONSTANT
	gParSaveMax						:UDINT:=20;
	gNoteArryMaxNum					:INT:=10;
	gRoughtPumVaccum				:REAL:=40.0;// mTorr
	gLoadLockPumSVaccum				:REAL:=90000.0;// mTorr
	gUltimateVacuum					:REAL:=5E-5;// 极限真空 Torr
	gATMPressure					:REAL:=740000.0;// 大气压力
	gATMPressureChamber				:REAL:=760000.0;// 大气压力
	gLVacuumPressureChamber			:REAL:=600.0;// 低气压 40mTorr以下
	gDifferentialPressure			:real:=300;
	gRFRFOffset						:UDINT:=5;
	gRFReflectPowerMin				:UDINT:=10;
	gMFCMonitParLimit				:UDINT:=1;
END_VAR

// ---- GVLs/GVL_AllGLOBAL.TcGVL
//{attribute 'qualified_only'}
VAR_GLOBAL
//结构体实例化
	gICP							:ST_ICP;// 结构体实例化
	
	
	gMachineUtility					:ST_MachineUtility;// 整机 面板IO
	MainFramDUT						:MainFram;//主框架参数绑定
	gCtrlMode						:ControlMode:=ControlMode.eManualCtrMode;//控制模式
	
//	gLoadModel						:ST_POUCommunication;
	
//	gLoadActPos						:ST_LoadActPos;//上料工作位，动作位置
//	gLoadDutState					:ST_HaveDUTState;//上料DUT状态
		
	SW1_PLC							:struct_Tester;//Sw1发往PLC信息结构体
//函数实例化
	gLog							:printLogModule_EX;// 用于打印运行 error log信息
	gDownTimeLog					:printLogModule_EX;// 用于打印运行 error log信息
	gDataChangeLog					:printLogModule_EX;// 用于打印 数据更改 运行log信息
	gBreakTimeLog					:printLogModule_EX;// 用于打印运行 BreakTime log信息
	gOperatorLog					:printLogModule_EX;// 操作日志
	gRunningLog						:printLogModule_EX;// 运行日志
	gShowPOURunLog					:BOOL;
	gShowLogTextTitle				:STRING;
	fb_systemTimeModule				:systemTimeModule;//获取系统时间
//Bool
	gsave							:BOOL;//配置保存按钮
	gSaveTemp						:BOOL;//配置保存中间变量
	gRead							:BOOL;//配置读取按钮
	gWindowsPageBt					: ARRAY [1..10] OF BOOL:=[TRUE];
	//机台系统变量
	gAutoRunningFlag				:BOOL:=FALSE;//自动运行中标志
	gErrorAbort						:BOOL;// ErrorAbort 退出半自动动作

	 // Recipe
	gRecipeNameSelect				:ARRAY [1..100] OF RecipeShowStr; 	// RecipeName
	gRecipeNameSelectShow			:ARRAY [1..10] OF RecipeShowStr; 	// RecipeName
	gRecipeFullPath					:STRING;	
	gRecipeShowNameOld				:STRING:='Recipe';
	gRecipeShowNameNow				:STRING;
	gRecipeEditorData				:ARRAY [1..gRecipeMAX_String_NUM] OF RecipePar; 
	gRecipeViewData					:ARRAY [1..gRecipeMAX_String_NUM] OF RecipePar;     
	gShowNum						:INT:=25;// Editor & View 显示的行数
	gselectRow						:INT:=0;// Recipe Editor 选取行号	
	gselectclo						:INT:=0;// Recipe Editor 选取列号	
	gRecipeSelctMaxIndex			:INT:=10;
	gRFSetTime						:UDINT;// 设置控制时间
	gRFRemainTime					:UDINT;// 剩余控制时间
	gRecipeSelectStruct				:ARRAY [1..gRecipeNameMAX_CSV_ROWS] OF RecipeNamePar;
	
	gRecipeSelectIndex1				:INT:=1;// Recipe选取的Index；方便探寻gRecipeSelect内部元素
	gRecipeNameMax					:UDINT:=1;// Recipe选取的Index；方便探寻gRecipeSelect内部元素
	gRFComControl					:BOOL;// RF双电源控制
	gWarmShowHMI					:WARMStruct;// showTrig
	gNoteShowHMI					:NoteStruct;// showTrig
	
	gRoughRemain					:BOOL;// 粗抽标记
	gRoughRemainTMPCanOpen			:BOOL;// 粗抽标记-运行开分子泵
	gSPOUBusy						:BOOL;// 任意一个程序在执行
	//TCPIP 网络变量
	gEnableSWConnect				:BOOL:=FALSE;//软件连接控制
	gEnablePDVSWConnect				:BOOL:=TRUE;//软件连接控制
	gEnableChillerSWConnect			:BOOL:=TRUE;//软件连接控制
	gEnableSRFSWConnect				:BOOL:=TRUE;//软件连接控制
	gEnablePRFSWConnect				:BOOL:=TRUE;//软件连接控制
	gEnableHeGSWConnect				:BOOL:=TRUE;//软件连接控制
	EnableAMXAISWConnect			:BOOL:=TRUE;//软件连接控制
	gEnableWaferCheck				:INT:=0;// 是否检测晶圆    0:不检测(提示框NO)；1：检测(提示框YES)；2：提示框弹出；
	
	gSWConnected					:BOOL;//主控
	gSWStringConnected				:BOOL;//主控
	gChillerConnected				:BOOL;//Chiller 
	gPDVConnected					:BOOL;//PDV 
	gSourceRFConnected				:BOOL;//SourceRF 
	gPowerRFConnected				:BOOL;//PowerRF 
	gHeliumGaugeConnected			:BOOL;//HeliumGauge 
	gAMXAIConnected					:BOOL;//艾莫迅AI模块 
	//所有软件连接
	gEnableSWConnectAll				:BOOL:=FALSE;//是否启用所有软件连接
	//机台所需临时调试变量
	gDisableSensor					:BOOL;
	gDisablePressureCheck			:BOOL;// 禁用压力检查
	gDisableWaterFloweCheck			:BOOL;// 禁用水流检查
	gDisableWaterTemCheck			:BOOL;// 禁用水压检查
	gEnablePDVOpenClose				:BOOL;// 强制启用PDV
	gEnableGDOpenClose				:BOOL;// 强制启用GateDoor
	gEnableHeInOpenClose			:BOOL;// 强制启用HeIn
	gPDVOpencondition				:BOOL;// PDV由关到开的检测条件
	gGDOpencondition				:BOOL;// GateDoor由关到开的检测条件
	gChamberVacRem					:REAL:=9000.0;// 腔体气压检测
	gTBVacRem						:REAL:=11000.0;// TB气压检测
	gCO_ControlRFTimeRemain			:UDINT:=0;
	
	gMFCStopLoopRead				:BOOL;// MFC读写锁：读优先级大于写优先级
	gTBPStopLoopRead				:BOOL;// TBP读写锁：读优先级大于写优先级
	
	gCNErrShow						:BOOL:=FALSE;//中英文切换显示
//Int
	//以太网
	gRemoteHostPort					:UINT:=5001;//远程连接端口
	gLocalHostPort					:UINT:=7920;//本地连接端口
	//时间转换配置变量
	gLoopTrgTime					:UDINT:=500;//循环触发相机时间设置
	gGetCCDResultTimeOut			:UDINT:=5000;//获取相机拍照结果超时时间
	//轴变量
	g_AxisOverride1					:LREAL:=100;
	gPosConfirm						:LREAL:=0.01;
	
	gCO_ControlRFRMTime				:UDINT:=0;		
//Real

//String
	g_sAmsNetId						:STRING;//获取arrAmsNetId
	g_SystemTime					:STRING;// Main 界面显示系统时间
	gVersion						:STRING:='V2.1.1.0';//进场版本
	gErrWTxtShow					:WSTRING(255):="";// Main 设备错误内容显示文本 中文---HMI
	gErrTxtShow						:STRING(255):='';// Main 设备错误内容显示文本---HMI
	gRemoteHostIp					:STRING:='192.168.1.200';//原创连接IP
	gLocalHostIp					:STRING:='192.168.1.100';//本地连接IP
	g_Test							:STRING:='10.0';// 测试使用
	g_Test1							:REAL;

//通讯变量
	gTxBuffer_SRF:					ComBuffer;// 顶部RF		
	gRxBuffer_SRF:					ComBuffer;// 底部RF
	
	gTxBuffer_MFC:					ComBuffer;// MFC		
	gRxBuffer_MFC:					ComBuffer;// MFC
	
	gTxBuffer_ARM:					ComBuffer;// MFC		
	gRxBuffer_ARM:					ComBuffer;// MFC
	
	gTxBuffer_TBP:					ComBuffer;// TBP		
	gRxBuffer_TBP:					ComBuffer;// TBP
// ADS命令交互
	gSTA2BData						:ST_A2BData;
	gSTB2AData						:ST_B2AData;
	gADSConnected					:BOOL;
	gTestBool						:BOOL;
	gTestInt						:INT;
	gTestReal						:REAL;
	gCurrentUser					:WSTRING;
	
	gPSGMaxPre_V					:REAL:=10.6635;// 模块压力校准
END_VAR

// ---- GVLs/GVL_AllPERSISTENT.TcGVL
//{attribute 'qualified_only'}
VAR_GLOBAL PERSISTENT
	gEnablePower					:BOOL:=TRUE;
	gWaferMemoryState				:INT:=0;// Charmber晶圆记忆状态    0:没有晶圆；1：有晶圆但未Etch； 2：有晶圆且Etch完成；
	gARMPosition					:DINT:=8900;// ARM 工作位	
	gCO_ControlRFTime				:UDINT:=10;		
END_VAR

// ---- GVLs/GVL_Datasave.TcGVL
//{attribute 'qualified_only'}
VAR_GLOBAL
//位置成组安全移动
	//上料相机轴
	DOEAXIS1AxisParSet				: ARRAY [1..20] OF ST_StationConfigBase;
	DOEAXIS2AxisParSet				: ARRAY [1..20] OF ST_StationConfigBase;
	//速度设置
	//临时采取用快速设置的方式
//	gStepAxisVel					:LREAL:=2.0;
//	gServoAxisVel					:LREAL:=20.0;

	
	gTestDelayTime: DINT;
	gDataArrName2					: ARRAY [1..20] OF WSTRING;// 20个点位名称
//DOE共轴界面参数设置
END_VAR
VAR_GLOBAL PERSISTENT
	;
END_VAR

// ---- POUs/BaseModule/ActionModule/GVL_ActionModule.TcGVL
//{attribute 'qualified_only'}
VAR_GLOBAL

END_VAR

// ---- POUs/BaseModule/DataSaveModule_EX/GVL_DataSave_EX.TcGVL
VAR_GLOBAL CONSTANT
	gMaxNumLength			: UDINT := 12800;//文件存储的字符最大容量  256000
	gNumBegin				: UDINT := 1;
END_VAR

VAR_GLOBAL CONSTANT
	(*这部分可按照实际项目去分配数量*)
	gMAX_BOOL_NUM			: UDINT := 179;//实际180
	gMAX_DINT_NUM			: UDINT := 179;//实际180
	gMAX_LREAL_NUM			: UDINT := 899;//实际899
	// Recipe
	gRecipeMAX_String_NUM	: UDINT := 22;//实际20
	gRecipeMAX_Show_Max		: UDINT := 20;
	
	gRecipeNameMAX_String_NUM	: UDINT := 99;//实际100
	gRecipeStepMaxShow:UDINT:=22;
END_VAR

VAR_GLOBAL CONSTANT
	gMAX_CSV_ROWS 			: UDINT := gMAX_BOOL_NUM + gMAX_DINT_NUM + gMAX_LREAL_NUM + 3;
	gMAX_CSV_COLUMNS 		: UDINT := 4;//实际有5列
	gMAX_CSV_FIELD_LENGTH	: UDINT := gMAX_BOOL_NUM + gMAX_DINT_NUM + gMAX_LREAL_NUM + 3;
	// Recipe
	gRecipeMAX_CSV_ROWS 		: UDINT := gRecipeMAX_String_NUM + 1;
	gRecipeMAX_CSV_COLUMNS 		: UDINT := 19;// 实际有20列
	gRecipeMAX_CSV_FIELD_LENGTH	: UDINT := gRecipeMAX_String_NUM + 1;
	
	gRecipeNameMAX_CSV_ROWS 		: UDINT := gRecipeNameMAX_String_NUM + 1;
	gRecipeNameMAX_CSV_COLUMNS 		: UDINT := 4;// 实际有20列
	gRecipeNameMAX_CSV_FIELD_LENGTH	: UDINT := gRecipeNameMAX_String_NUM + 1;
END_VAR

// ---- POUs/BaseModule/Error/GVL_Error.TcGVL
//{attribute 'qualified_only'}
VAR_GLOBAL CONSTANT
	g_d_ErrorBegin		:DINT:=0;
	g_d_ErrorEnd		:DINT:=8000;
	g_Max_Data_Elements :UDINT:=100;(* Max. number of elements in the list *)
END_VAR
VAR_GLOBAL
	gErrorARRAY	:ARRAY [g_d_ErrorBegin..g_d_ErrorEnd] OF ST_Error;
	
	gError_fbTable:FB_HashTableCtrl;(* basic hash table control function block *)
    gError_hTable:T_HHASHTABLE;(* hash table handle *)
    gError_table:ARRAY[0..g_Max_Data_Elements] OF T_HashTableEntry;
END_VAR

// ---- POUs/BaseModule/PrintLogModule_EX/GVL_PrintLogModule_EX.TcGVL
//{attribute 'qualified_only'}
VAR_GLOBAL CONSTANT
	cNumLength				:DINT:=256;			//log堆栈保存的最大数量
	cNumBegin				:DINT:=1;			//默认为 1
	cNumLength_showInof		:DINT:=100;			//默认显示 100 记录
	cNumBegin_showInof		:DINT:=1;			//默认为 1
END_VAR

// ---- POUs/BaseModule/SystemTimeModule/GVL_SystemTimeModule.TcGVL
//{attribute 'qualified_only'}
VAR_GLOBAL
END_VAR
VAR_GLOBAL CONSTANT
	gSystemTimeMaxNum		:UINT:=2000;// systemTimeModule 计时器数组最大值 最大值为2000
END_VAR

// ---- POUs/BaseModule/TcpIpModule_EX/GVL_TcpIpModule_EX.TcGVL
//{attribute 'qualified_only'}
VAR_GLOBAL CONSTANT
	(*这部分可按照实际项目去分配数量*)
	g_nMaxByte_Client			:UINT:=32;//二进制数据结构字符最大长度
	g_nMaxByte_Server			:UINT:=32;//二进制数据结构字符最大长度
END_VAR

VAR_GLOBAL
	
END_VAR

// ---- POUs/Other/MachineState/GVL_MachineState.TcGVL
//{attribute 'qualified_only'}
VAR_GLOBAL
	fbMachineState		:FB_MachineState;
	gRunningState		:RunningStatus:=RunningStatus.eManualState;
END_VAR

// ---- POUs/Other/ActBase/ITF/ITFActStep.TcIO
(*
---Control step base interface
*)
INTERFACE ITFActStep

(*
---Continue action
*)
METHOD Act_Continue : BOOL
VAR_INPUT
END_VAR
END_METHOD

(*
---Trigger action
*)
METHOD Act_Ex : BOOL
VAR_INPUT
END_VAR
END_METHOD

(*
---Init all status
*)
METHOD Act_Init : BOOL
VAR_INPUT
END_VAR
END_METHOD

(*
---Pause action
*)
METHOD Act_Pause : BOOL
VAR_INPUT
	pause:BOOL;
END_VAR
END_METHOD

(*
---: add step;
---:
	nextStep: step 增量值;
	checkPause: 是否检测当前 pause; 如果 checkPause:=TRUE, 且暂停被触发后, 当前 step 暂停递增;
*)
METHOD addStep : DINT
VAR_INPUT
	nextStep			:DINT:=0;
	checkPause			:BOOL:=FALSE;// 检查是否暂停，暂停则不递增step
END_VAR
END_METHOD

(*
---Get action state
*)
METHOD getActState : ST_ActStep_State
VAR_INPUT
END_VAR
END_METHOD

(*
---Get error id
*)
METHOD getErrID : DINT
VAR_INPUT
END_VAR
END_METHOD

(*
---Get error message
*)
METHOD getErrMsg : STRING(255)
VAR_INPUT
END_VAR
END_METHOD

(*
---Get error step
*)
METHOD getErrStep : DINT
VAR_INPUT
END_VAR
END_METHOD

(*
---Get step
*)
METHOD getStep : DINT
VAR_INPUT
END_VAR
END_METHOD

(*
---Check busy state
*)
METHOD isBusy : BOOL
VAR_INPUT
END_VAR
END_METHOD

(*
---Check done state
*)
METHOD isDone : BOOL
VAR_INPUT
END_VAR
END_METHOD

(*
---Check error state
*)
METHOD isError : BOOL
VAR_INPUT
END_VAR
END_METHOD

(*
---Check trigger state
*)
METHOD isEx : BOOL
VAR_INPUT
END_VAR
END_METHOD

(*
---Check pause state
*)
METHOD isPause : BOOL
VAR_INPUT
END_VAR
END_METHOD

(*
---Set busy flag
*)
METHOD setBusyFlag
VAR_INPUT
END_VAR
END_METHOD

(*
---Set done flag
*)
METHOD setDoneFlag
VAR_INPUT
END_VAR
END_METHOD

(*
---Set error done flag
*)
METHOD setErrDoneFlag
VAR_INPUT
END_VAR
END_METHOD

(*
---Set error id
*)
METHOD setErrID
VAR_INPUT
	errID:DINT;
END_VAR
END_METHOD

(*
---Set error message
*)
METHOD setErrMsg
VAR_INPUT
	errMsg:STRING(255);
END_VAR
END_METHOD

(*
---Set error id and error message
*)
METHOD setError
VAR_INPUT
	errID:DINT;
	errMsg:STRING(255);
END_VAR
END_METHOD

(*
---Go to step:=BEGIN_STEP, BEGIN_STEP is 10;
*)
METHOD toBeginStep : DINT
VAR_INPUT
END_VAR
END_METHOD

(*
---Go to step:=DONE_STEP, DONE_STEP is 60000;
*)
METHOD toDoneStep : DINT
VAR_INPUT
END_VAR
END_METHOD

(*
---Go to step:=ERR_DONE_STEP, ERR_DONE_STEP is 65000;
*)
METHOD toErrDoneStep : DINT
VAR_INPUT
END_VAR
END_METHOD

(*
---Go to pause step:=PAUSE_STEP, PAUSE_STEP is 65500; 
---: nextStep: 从暂停解除之后的下一个step值; 
*)
METHOD toPauseStep : DINT
VAR_INPUT
	{attribute 'initialize_on_call'}
	nextStep			:DINT:=0;
END_VAR
END_METHOD

(*
---: Go to target step;
---:
	nextStep: step 目标值;
	checkPause: 是否检测当前 pause; 如果 checkPause:=TRUE, 且暂停被触发后, 当前 step 暂停递增;
*)
METHOD toStep : DINT
VAR_INPUT
	nextStep			:DINT:=0;// 跳转到目标step
	checkPause			:BOOL:=FALSE;// 检查是否暂停，暂停则不递增step
END_VAR
END_METHOD

(*
---Go to step:=0;
*)
METHOD toZeroStep : DINT
VAR_INPUT
END_VAR
END_METHOD

END_INTERFACE

// ---- POUs/Other/ActBase/ITF/ITFUserAction.TcIO
INTERFACE ITFUserAction

(*
---Abort action
*)
METHOD Act_Abort : BOOL
VAR_INPUT
END_VAR
END_METHOD

(*
---Continue action
*)
METHOD Act_Continue : BOOL
VAR_INPUT
END_VAR
END_METHOD

(*
---Trigger action
*)
METHOD Act_Ex : BOOL
VAR_INPUT
END_VAR
END_METHOD

(*
---Init all status
*)
METHOD Act_Init : BOOL
VAR_INPUT
END_VAR
END_METHOD

(*
---Pause action
*)
METHOD Act_Pause : BOOL
VAR_INPUT
	pause:BOOL;
END_VAR
END_METHOD

(*
---Reset Action
*)
METHOD Act_Reset : BOOL
VAR_INPUT
END_VAR
END_METHOD

(*
---Stop action
*)
METHOD Act_Stop : BOOL
VAR_INPUT
END_VAR
END_METHOD

(*
---Get busy signal
*)
METHOD Get_Busy : BOOL
VAR_INPUT
END_VAR
END_METHOD

(*
---Get done signal
*)
METHOD Get_Done : BOOL
VAR_INPUT
END_VAR
END_METHOD

(*
---Get error signal
*)
METHOD Get_Error : BOOL
VAR_INPUT
END_VAR
END_METHOD

END_INTERFACE

// ---- POUs/Communication/RS232_485_ALLEL.TcPOU
PROGRAM RS232_485_ALLEL
VAR
	(*
	 *xBuffer 的作用是，在 PLC 要发送的数据和串行通讯的硬件 Process Data 之间设置一个缓存区。
	 *比如 KL6outData22B 类型的接口，每个 PLC 周期只能发送 22 字节。假如程序需要发送的数据为 100 个，
	 *那么实际上 PLC 程序是把这些数据放到 TxBuffer 中，再由硬件分几个 PLC 周期发送出去
	*)

	SRF_COMin				AT%I*		:KL6inData22B;		
	SRF_COMout				AT%Q*		:KL6outData22B;
	SRF_Error				:BOOL;
		
	SRF_COMportControl					:SerialLineControl;
	
	MFC_COMin				AT%I*		:KL6inData22B;		
	MFC_COMout				AT%Q*		:KL6outData22B;
	MFC_Error				:BOOL;
		
	MFC_COMportControl					:SerialLineControl;
	
	ARM_COMin				AT%I*		:KL6inData22B;		
	ARM_COMout				AT%Q*		:KL6outData22B;
	ARM_Error				:BOOL;
		
	ARM_COMportControl					:SerialLineControl;
	
	TBP_COMin				AT%I*		:KL6inData22B;		
	TBP_COMout				AT%Q*		:KL6outData22B;
	TBP_Error				:BOOL;
		
	TBP_COMportControl					:SerialLineControl;
	
END_VAR

(*
 *功能块的作用，把 TxBuffer 缓存区的数据经过 Process Data 的 ComOut 发送出去，
 *而把 ComIn 中的数据接收到 RxBuffer。引用这个功能块的程序执行周期越短，
 *数据交换的效率就越高，所以这段程序应该放在快速任务中作为 Backgroud 代码无条件执行。
*)
SRF_COMportControl(
	Mode:= SERIALLINEMODE_KL6_22B_STANDARD, 
	pComIn:= ADR(SRF_COMin), 
	pComOut:= ADR(SRF_COMout), 
	SizeComIn:= SIZEOF(SRF_COMin), 
	Error=> , 
	ErrorID=> , 
	TxBuffer:= gTxBuffer_SRF, 
	RxBuffer:= gRxBuffer_SRF );
IF SRF_COMportControl.Error THEN
	SRF_Error:=TRUE;
ELSE
	SRF_Error:=FALSE;
END_IF

MFC_COMportControl(
	Mode:= SERIALLINEMODE_KL6_22B_STANDARD, 
	pComIn:= ADR(MFC_COMin), 
	pComOut:= ADR(MFC_COMout), 
	SizeComIn:= SIZEOF(MFC_COMin), 
	Error=> , 
	ErrorID=> , 
	TxBuffer:= gTxBuffer_MFC, 
	RxBuffer:= gRxBuffer_MFC );
IF MFC_COMportControl.Error THEN
	MFC_Error:=TRUE;
ELSE
	MFC_Error:=FALSE;
END_IF

ARM_COMportControl(
	Mode:= SERIALLINEMODE_KL6_22B_STANDARD, 
	pComIn:= ADR(ARM_COMin), 
	pComOut:= ADR(ARM_COMout), 
	SizeComIn:= SIZEOF(ARM_COMin), 
	Error=> , 
	ErrorID=> , 
	TxBuffer:= gTxBuffer_ARM, 
	RxBuffer:= gRxBuffer_ARM );
IF ARM_COMportControl.Error THEN
	ARM_Error:=TRUE;
ELSE
	ARM_Error:=FALSE;
END_IF

TBP_COMportControl(
	Mode:= SERIALLINEMODE_KL6_22B_STANDARD, 
	pComIn:= ADR(TBP_COMin), 
	pComOut:= ADR(TBP_COMout), 
	SizeComIn:= SIZEOF(TBP_COMin), 
	Error=> , 
	ErrorID=> , 
	TxBuffer:= gTxBuffer_TBP, 
	RxBuffer:= gRxBuffer_TBP );
IF TBP_COMportControl.Error THEN
	TBP_Error:=TRUE;
ELSE
	TBP_Error:=FALSE;
END_IF

END_PROGRAM

// ---- POUs/Data/DataSave.TcPOU
PROGRAM DataSave
VAR_INPUT
	fbDataSaveModule_EX_1			:DataSaveModule_EX;
	fbDataSaveModule_EX_recipe		:RecipeSaveModule_EX;
	fbDataSaveModule_EX_recipename	:RecipeNameModule_EX;
	RecipeDataClear					:ARRAY [1..gRecipeMAX_String_NUM] OF RecipePar;     
	//上料相机轴
	DOEX1AxisPar					: ARRAY [1..20] OF FB_SavePar;
	DOEX2AxisPar					: ARRAY [1..20] OF FB_SavePar;
	wstrShow						:WSTRING:="";
END_VAR
VAR_OUTPUT
	busy					:BOOL;
	done					:BOOL;
	error					:BOOL;
END_VAR
VAR
	itemp:INT;
	jtemp:INT;
	save_R_Trig				:R_Trig;
	load_R_Trig				:R_Trig;
	
	save_F_Trig				:F_Trig;
	load_F_Trig				:F_Trig;
	chinnesename			:WSTRING;
	posname					:WSTRING;
	englishname				:STRING;
	
//	rtrig_RX				:R_TRIG;
	error_Rtrig				:R_TRIG;
END_VAR
VAR
	
	
END_VAR
VAR
	nSaveStep:INT;
	tTimeout:TON;
	stamovestep:INT;
	
	tLoadTime:TON;
	TestRead:LREAL;	
	RXPosIndex : UINT;
END_VAR


//
fbDataSaveModule_EX_recipe.RecipeChange();
save_R_Trig(CLK:=gSaveTemp OR gsave );//点击保存按钮:需要并上某一条件，进行限制
//rtrig_RX(CLK:=gDUTType=0 , Q=> );

//IF rtrig_TX.Q THEN
//	gRead:=TRUE;
//END_IF

//
IF save_R_Trig.Q THEN
	gLog.append('Save All Config');
	gDataChangeLog.append_EX("数据发生更改");
	gSaveTemp:=FALSE;
	ups_CX51X0.Act_Wrtie();
	IF 0=nSaveStep THEN
		nSaveStep:=100;
	END_IF
END_IF
load_R_Trig(CLK:=gRead);

tLoadTime(IN:= gRead, PT:=T#1S , Q=> , ET=> );
load_F_Trig(CLK:=tLoadTime.Q , Q=> );
//


IF load_R_Trig.Q THEN
	gDataChangeLog.append_EX(" DOE 配置");
	gLog.append('Load All Config');
	fbDataSaveModule_EX_1.readB:=TRUE;//按实际需要进行屏蔽和启用
	fbDataSaveModule_EX_recipe.readB:=TRUE;
END_IF
error_Rtrig(CLK:=NOT MainRunPOU.DelayFlag AND fbDataSaveModule_EX_recipe.error AND 
				 fbDataSaveModule_EX_recipe.checkFileExistError AND NOT fbDataSaveModule_EX_recipe.busy, Q=> );
IF error_Rtrig.Q  THEN
	gShowNum:=0;
	gRecipeEditorData:=RecipeDataClear;
	gRecipeViewData:=RecipeDataClear;
	
	gLog.append(gRecipeShowNameNow);
	error_Trigger(30);
END_IF

ACT_MainPara();
ACT_StructInstance_DOE();



busy:=fbDataSaveModule_EX_1.busy    //按实际需要进行屏蔽和启用
		;
error:=fbDataSaveModule_EX_1.error  //按实际需要进行屏蔽和启用
		;

tTimeout(IN:=0<>nSaveStep,PT:=T#10S);
IF tTimeout.Q THEN
	tTimeout(IN:=FALSE);
	nSaveStep:=0;
END_IF
CASE nSaveStep OF
	0:
		;
	100:
		IF NOT fbDataSaveModule_EX_1.busy THEN
			nSaveStep:=nSaveStep+10;
		END_IF
	110:
		//savePara1_Inner:=TRUE;
		nSaveStep:=nSaveStep+10;
	120:
		IF fbDataSaveModule_EX_1.busy THEN
			nSaveStep:=nSaveStep+10;
		END_IF
	130:
		IF NOT fbDataSaveModule_EX_1.busy THEN
			nSaveStep:=nSaveStep+10;
		END_IF
	140:
		nSaveStep:=500;
		
	500:
		nSaveStep:=0;
END_CASE

ACTION ACT_MainPara:

//(*
//保存参数


IF save_R_Trig.Q THEN
	gLog.append('Save Sta1 Config');
	
	//offset-500-720
//Int类型存储

	
	
	fbDataSaveModule_EX_1.setDintValue((gTestDelayTime),4);
//	fbDataSaveModule_EX_1.setDintValue((gDUTType),5);
	
//	fbDataSaveModule_EX_1.setBoolValue((gTXPosEnable[0]),10);
//	fbDataSaveModule_EX_1.setBoolValue((gTXPosEnable[1]),11);
//	fbDataSaveModule_EX_1.setBoolValue((gTXPosEnable[2]),12);
//	fbDataSaveModule_EX_1.setBoolValue((gTXPosEnable[3]),13);
//	fbDataSaveModule_EX_1.setBoolValue((gTXPosEnable[4]),14);
//	fbDataSaveModule_EX_1.setBoolValue((gTXPosEnable[5]),15);
//	fbDataSaveModule_EX_1.setBoolValue((gTXPosEnable[6]),16);
//	fbDataSaveModule_EX_1.setBoolValue((gTXPosEnable[7]),17);
	
//	fbDataSaveModule_EX_1.setBoolValue(gEnableCOffset,20); 
//	fbDataSaveModule_EX_1.setBoolValue(gEnableTxOffset,21); 
//	fbDataSaveModule_EX_1.setBoolValue(gEnableRXLimit,22); 
//	fbDataSaveModule_EX_1.setBoolValue(gEnableRXOffset,23); 
	

 	fbDataSaveModule_EX_1.setLrealValue(FuncModule_RS232_SRF.goPosLoad,1);
	fbDataSaveModule_EX_1.setLrealValue(FuncModule_RS232_SRF.goPosPhase,2);
	
//中文文档读写
	FB_WStringSave.setWString(gDataArrName2[1],1);
	FB_WStringSave.setWString(gDataArrName2[2],2);
	FB_WStringSave.setWString(gDataArrName2[3],3);
	FB_WStringSave.setWString(gDataArrName2[4],4);
	FB_WStringSave.setWString(gDataArrName2[5],5);
	FB_WStringSave.setWString(gDataArrName2[6],6);
	FB_WStringSave.setWString(gDataArrName2[7],7);
	FB_WStringSave.setWString(gDataArrName2[8],8);
	FB_WStringSave.setWString(gDataArrName2[9],9);
	FB_WStringSave.setWString(gDataArrName2[10],10);
	FB_WStringSave.setWString(gDataArrName2[11],11);
	FB_WStringSave.setWString(gDataArrName2[12],12);
	FB_WStringSave.setWString(gDataArrName2[13],13);
	FB_WStringSave.setWString(gDataArrName2[14],14);
	FB_WStringSave.setWString(gDataArrName2[15],15);
	FB_WStringSave.setWString(gDataArrName2[16],16);
	FB_WStringSave.setWString(gDataArrName2[17],17);
	FB_WStringSave.setWString(gDataArrName2[18],18);
	FB_WStringSave.setWString(gDataArrName2[19],19);
	FB_WStringSave.setWString(gDataArrName2[20],20);
	FB_WStringSave.writeTrig:=TRUE;
	fbDataSaveModule_EX_1.saveB:=TRUE;
	fbDataSaveModule_EX_recipe.saveB:=TRUE;
	ups_CX51X0.Act_Wrtie();
END_IF
//*)
//(*
//读取参数
IF tLoadTime.Q AND DataSave.fbDataSaveModule_EX_recipe.rDone THEN
	fbDataSaveModule_EX_recipe.readB:=FALSE;
END_IF


IF tLoadTime.Q AND DataSave.fbDataSaveModule_EX_1.rDone THEN

//Int类型存储
	
	fbDataSaveModule_EX_1.getDintValue((gTestDelayTime),4);
//	fbDataSaveModule_EX_1.getDintValue((gDutTypeComfirm),5);
	
//	fbDataSaveModule_EX_1.getBoolValue((gTXPosEnable[0]),10);
//	fbDataSaveModule_EX_1.getBoolValue((gTXPosEnable[1]),11);
//	fbDataSaveModule_EX_1.getBoolValue((gTXPosEnable[2]),12);
//	fbDataSaveModule_EX_1.getBoolValue((gTXPosEnable[3]),13);
//	fbDataSaveModule_EX_1.getBoolValue((gTXPosEnable[4]),14);
//	fbDataSaveModule_EX_1.getBoolValue((gTXPosEnable[5]),15);
//	fbDataSaveModule_EX_1.getBoolValue((gTXPosEnable[6]),16);
//	fbDataSaveModule_EX_1.getBoolValue((gTXPosEnable[7]),17);
	
//	fbDataSaveModule_EX_1.getBoolValue(gEnableCOffset,20);
//	fbDataSaveModule_EX_1.getBoolValue(gEnableTxOffset,21); 
//	fbDataSaveModule_EX_1.getBoolValue(gEnableRXLimit,22); 
//	fbDataSaveModule_EX_1.getBoolValue(gEnableRXOffset,23); 
////上料速度
// 	fbDataSaveModule_EX_1.getLrealValue(gLoad_AXIS.Y1RunVel,600);
//	fbDataSaveModule_EX_1.getLrealValue(gLoad_AXIS.X1RunVel,601);
//	fbDataSaveModule_EX_1.getLrealValue(gLoad_AXIS.Z1RunVel,602);
//	fbDataSaveModule_EX_1.getLrealValue(gLoad_AXIS.R1RunVel,603);
//	fbDataSaveModule_EX_1.getLrealValue(gLoad_AXIS.CY1RunVel,604);
//	fbDataSaveModule_EX_1.getLrealValue(gUnLoad_AXIS.CY1RunVel,605);

	fbDataSaveModule_EX_1.getLrealValue(FuncModule_RS232_SRF.goPosLoad,1);
	fbDataSaveModule_EX_1.getLrealValue(FuncModule_RS232_SRF.goPosPhase,2);	


	fbDataSaveModule_EX_1.readB:=FALSE;
	gRead:=FALSE;
END_IF
IF load_F_Trig.Q THEN
	FB_WStringSave.readTrig:=TRUE;
END_IF
IF FB_WStringSave.readDone THEN
	FB_WStringSave.getWString(gDataArrName2[1],1);
	FB_WStringSave.getWString(gDataArrName2[2],2);
	FB_WStringSave.getWString(gDataArrName2[3],3);
	FB_WStringSave.getWString(gDataArrName2[4],4);
	FB_WStringSave.getWString(gDataArrName2[5],5);
	FB_WStringSave.getWString(gDataArrName2[6],6);
	FB_WStringSave.getWString(gDataArrName2[7],7);
	FB_WStringSave.getWString(gDataArrName2[8],8);
	FB_WStringSave.getWString(gDataArrName2[9],9);
	FB_WStringSave.getWString(gDataArrName2[10],10);
	FB_WStringSave.getWString(gDataArrName2[11],11);
	FB_WStringSave.getWString(gDataArrName2[12],12);
	FB_WStringSave.getWString(gDataArrName2[13],13);
	FB_WStringSave.getWString(gDataArrName2[14],14);
	FB_WStringSave.getWString(gDataArrName2[15],15);
	FB_WStringSave.getWString(gDataArrName2[16],16);
	FB_WStringSave.getWString(gDataArrName2[17],17);
	FB_WStringSave.getWString(gDataArrName2[18],18);
	FB_WStringSave.getWString(gDataArrName2[19],19);
	FB_WStringSave.getWString(gDataArrName2[20],20);
	;
END_IF

//*)
//其他
fbDataSaveModule_EX_1(
		sFileName:= 'C:\Config\ICP_Para.csv', 
		readB:= , 
		saveB:= , 
		dataBool:= , 
		dataBoolLength:= 50, 
		dataDint:= , 
		dataDintLength:= 50, 
		dataLreal:= , 
		dataLrealLength:=1000 , 
		busy=> , 
		rDone=> , 
		sDone=> , 
		error=> , 
		errID=> , 
		errTxt=> );
		
fbDataSaveModule_EX_recipename(
	sFileName:= 'C:\Config\Name.csv', 
	readB:= , 
	saveB:= , 
	dataString:= , 
	dataStringLength:=99 , 
	busy=> , 
	rDone=> , 
	sDone=> , 
	error=> , 
	errID=> , 
	errTxt=> );

gRecipeFullPath:='';
gRecipeFullPath:=CONCAT(gRecipeFullPath,'C:\Config\');
gRecipeFullPath:=CONCAT(gRecipeFullPath,gRecipeNameSelect[gRecipeSelectIndex1].Name);
gRecipeFullPath:=CONCAT(gRecipeFullPath,'.csv');
fbDataSaveModule_EX_recipe(
	sFileName:= gRecipeFullPath, 
	readB:= , 
	saveB:= , 
	dataString:= , 
	dataStringLength:= , 
	busy=> , 
	rDone=> , 
	sDone=> , 
	error=> , 
	errID=> , 
	errTxt=> );

FB_WStringSave(//中文读写
	filter:="," , 
	savePath:='C:\Config\ChinessPar.txt', 
	nErrorId=> , 
	bError=> , 
	readDone=> , 
	saveDone=> , 
	readError=> , 
	saveError=> );


fbDataSaveModule_EX_1.saveB:=FALSE;
fbDataSaveModule_EX_recipe.saveB:=FALSE;
END_ACTION

ACTION ACT_StructInstance_DOE:

////saveIndexOffset处于递增的过程

////offset-gParSaveMax倍数  0-5倍
//FOR itemp:=1 TO 20 BY 1 DO//相机景深CY1
	
//	chinnesename:=wCONCAT(chinnesename,"DOEAXIS1-");
//	chinnesename:=wCONCAT(chinnesename,gDataArrName2[itemp]);
//	englishname:=CONCAT(englishname,'DOEAXIS1 Parameter');
//	englishname:=CONCAT(englishname,TO_STRING(iTemp));
//	DOEAXIS1AxisParSet[itemp].RunVel:=gDOE_AXIS.DOE1RunVel;
//	IF gCNErrShow THEN
//		posname:=wCONCAT(posname,"位置");
//	ELSE
//		posname:=wCONCAT(posname,"Pos");
//	END_IF
//	posname:=wCONCAT(posname,TO_WSTRING(iTemp));
//	DOEX1AxisPar[itemp](////////
//		logOut:=gDataChangeLog,
//		gStaParSet:=DOEAXIS1AxisParSet[itemp] , ///////
//		motorAix:=gDOE_AXIS.DOE1Axis , 
//		saveRef:= fbDataSaveModule_EX_1, 
//		chinnesename:=chinnesename , ///////
//		pos1name:=posname,////
//		eglishname:= englishname,///// 
//		languageswitch:=gCNErrShow , 
//		saveIndexOffset:=0*20+itemp,///////
//		moveerro=> DOEAXIS1AxisParSet[itemp].moveerror, ////////
//		movebusy=> , 
//		movedone=> );
//	chinnesename:="";
//	posname:="";
//	englishname:='';
//END_FOR
//FOR itemp:=1 TO 20 BY 1 DO//相机景深CY1
//	chinnesename:=wCONCAT(chinnesename,"DOEAXIS2-");
//	chinnesename:=wCONCAT(chinnesename,gDataArrName2[itemp]);
//	englishname:=CONCAT(englishname,'DOEAXIS2 Parameter');
//	englishname:=CONCAT(englishname,TO_STRING(iTemp));
//	DOEAXIS2AxisParSet[itemp].RunVel:=gDOE_AXIS.DOE2RunVel;
//	IF gCNErrShow THEN
//		posname:=wCONCAT(posname,"位置");
//	ELSE
//		posname:=wCONCAT(posname,"Pos");
//	END_IF
//	posname:=wCONCAT(posname,TO_WSTRING(iTemp));
//	DOEX2AxisPar[itemp](////////
//		logOut:=gDataChangeLog,
//		gStaParSet:=DOEAXIS2AxisParSet[itemp] , ///////
//		motorAix:=gDOE_AXIS.DOE2Axis , 
//		saveRef:= fbDataSaveModule_EX_1, 
//		chinnesename:=chinnesename , ///////
//		pos1name:=posname,////
//		eglishname:= englishname,///// 
//		languageswitch:=gCNErrShow , 
//		saveIndexOffset:=1*20+itemp,///////
//		moveerro=> DOEAXIS2AxisParSet[itemp].moveerror, ////////
//		movebusy=> , 
//		movedone=> );
//	chinnesename:="";
//	posname:="";
//	englishname:='';
//END_FOR
END_ACTION

END_PROGRAM

// ---- POUs/BaseModule/DataSaveModule_EX/DataSaveModule_EX.TcPOU
FUNCTION_BLOCK DataSaveModule_EX
VAR_INPUT
	sFileName						:T_MaxString:='C:\IASaveData.csv';//'Hard Disk\IASaveData.csv'  数据文件存储路径
	readB							:BOOL:=FALSE;//读取触发
	saveB							:BOOL:=FALSE;//保存触发
	dataBool						:ARRAY[0..gMAX_BOOL_NUM] OF BOOL;//BOOL数据源
	dataBoolLength					:UDINT:=gMAX_BOOL_NUM;//BOOL数据源 长度，从0开始计数，且不能随意变动
	dataDint						:ARRAY[0..gMAX_DINT_NUM] OF DINT;//DINT数据源
	dataDintLength					:UDINT:=gMAX_DINT_NUM;//DINT数据源 长度，从0开始计数，且不能随意变动
	dataLreal						:ARRAY[0..gMAX_LREAL_NUM] OF LREAL;//LREAL数据源
	dataLrealLength					:UDINT:=gMAX_LREAL_NUM;//LREAL数据源 长度，从0开始计数，且不能随意变动
END_VAR
VAR_OUTPUT
	busy							:BOOL:=FALSE;
	rDone							:BOOL:=FALSE;
	sDone							:BOOL:=FALSE;
	error							:BOOL:=FALSE;
	errID							:UDINT:=0;
	errTxt							:STRING(255):='';
END_VAR
VAR_IN_OUT
	
END_VAR
VAR
	pDatabase						:ARRAY[0..gMAX_CSV_ROWS, 0..gMAX_CSV_COLUMNS ] OF STRING(30);(* Target PLC database *)	
	csv_rows						:UDINT:=gMAX_CSV_ROWS;
	csv_columns						:UDINT:=gMAX_CSV_COLUMNS;
	
	startUpB						:BOOL:=FALSE;
	writeTxt						:P_TextModeWrite;
	readTxt							:P_TextModeRead;
	fbFileOpen						:FB_FileOpen;//检查文件是否存在
	fbFileClose						:FB_FileClose;(* Closes file *)
	hFile							:UINT:=0;(* File handle of the source file *)
	checkFileExistError				:BOOL;
	initB							:BOOL:=FALSE;
	saveStep						:UINT:=0;
	readStep						:UINT:=0;
	sFileNameOld					:T_MaxString;//旧文件名
//获取系统时间
	ntGetTime				: NT_GetTime;
	systemTimeStruct		: TIMESTRUCT;
	getSystemTimeStep		: UINT:=0;
	systemTIMEStr			: STRING:='';//系统时间，格式YYYY-MM-DD hh:mm:ss_zzz
	systemTIMEStr2			: STRING:='';//系统时间，格式YYYYMMDDhhmmss
	sysTIMEStrYY			: STRING:='';//系统时间，年
	sysTIMEStrMM			: STRING:='';//系统时间，月
	sysTIMEStrDD			: STRING:='';//系统时间，日
	sysTIMEStr_HH			: STRING:='';//系统时间，时
	sysTIMEStr_mm			: STRING:='';//系统时间，分
	sysTIMEStr_ss			: STRING:='';//系统时间，秒
END_VAR

IF dataBoolLength>gMAX_BOOL_NUM THEN
	dataBoolLength:=gMAX_BOOL_NUM;
END_IF
IF dataDintLength>gMAX_DINT_NUM THEN
	dataDintLength:=gMAX_DINT_NUM;
END_IF
IF dataLrealLength>gMAX_LREAL_NUM THEN
	dataLrealLength:=gMAX_LREAL_NUM;
END_IF

csv_rows:=dataBoolLength + dataDintLength + dataLrealLength + 3;
IF csv_rows>gMAX_CSV_ROWS THEN
	csv_rows:=gMAX_CSV_ROWS;
END_IF

//judge length
IF gMAX_CSV_ROWS<(gMAX_BOOL_NUM+gMAX_DINT_NUM+gMAX_LREAL_NUM+3) THEN
	error:=TRUE;
	errTxt:='dataBase$'s length too short';
	RETURN;
END_IF
IF csv_rows<(dataBoolLength+dataDintLength+dataLrealLength+3) THEN
	error:=TRUE;
	errTxt:='dataBase$'s length too short';
	RETURN;
END_IF

init();
IF initB THEN
	readMethod();
	saveMethod();
END_IF
getSystemTime();

METHOD PRIVATE createDir : BOOL
VAR
	sPathNameTemp	: T_MaxString := 'C:\TwinCAT\Data.txt';
	sDriveTemp		: STRING(3);
	sDirTemp		: T_MaxString;
	sFileNameTemp	: T_MaxString;
	sExtTemp		: T_MaxString;
	bSuccess		: BOOL;
	fbCreateDir		: FB_CreateDir;
	fbCreateDir2		: FB_CreateDir;
	sFileDirTemp	: T_MaxString;
	sFileDirTemp2	: T_MaxString;
END_VAR
sPathNameTemp:=sFileName;
bSuccess := F_SplitPathName( sPathName := sPathNameTemp,
	sDrive := sDriveTemp,
	sDir := sDirTemp,
	sFileName := sFileNameTemp,
	sExt := sExtTemp );
IF bSuccess THEN
	bSuccess:=FALSE;
	IF LEFT(sDirTemp,LEN(sDirTemp)-1) <> '' THEN
		//sFileDirTemp:=CONCAT(STR1:=sDriveTemp,STR2:=LEFT(sDirTemp,LEN(sDirTemp)-1));
		//sFileNameOld:=CONCAT(STR1:=sFileDirTemp,STR2:=CONCAT('\',CONCAT(sFileNameTemp,'_Old.csv')));//用于重命名参数文件
		sFileDirTemp:='';
		sFileDirTemp:=CONCAT(sFileDirTemp,sDriveTemp);
		sFileDirTemp:=CONCAT(sFileDirTemp,LEFT(sDirTemp,LEN(sDirTemp)-1));
		sFileDirTemp2:='';
		sFileDirTemp2:=CONCAT(sFileDirTemp2,sFileDirTemp);
		sFileDirTemp2:=CONCAT(sFileDirTemp2,'\Old');
		
		sFileNameOld:='';
		sFileNameOld:=CONCAT(sFileNameOld,sFileDirTemp);
		sFileNameOld:=CONCAT(sFileNameOld,'\Old\');//'\'
		sFileNameOld:=CONCAT(sFileNameOld,sFileNameTemp);
		sFileNameOld:=CONCAT(sFileNameOld,'_Old_');
		sFileNameOld:=CONCAT(sFileNameOld,systemTIMEStr2);
		sFileNameOld:=CONCAT(sFileNameOld,'.csv');
		
		fbCreateDir(
			sNetId:= , 
			sPathName:= sFileDirTemp, 
			ePath:= PATH_GENERIC, 
			bExecute:= TRUE, 
			tTimeout:= , 
			bBusy=> , 
			bError=> , 
			nErrId=> );
		fbCreateDir2(
			sNetId:= , 
			sPathName:= sFileDirTemp2, 
			ePath:= PATH_GENERIC, 
			bExecute:= TRUE, 
			tTimeout:= , 
			bBusy=> , 
			bError=> , 
			nErrId=> );
	END_IF
END_IF
fbCreateDir(
	sNetId:= , 
	sPathName:= , 
	ePath:= , 
	bExecute:= FALSE, 
	tTimeout:= , 
	bBusy=> , 
	bError=> , 
	nErrId=> );
fbCreateDir2(
	sNetId:= , 
	sPathName:= , 
	ePath:= , 
	bExecute:= FALSE, 
	tTimeout:= , 
	bBusy=> , 
	bError=> , 
	nErrId=> );
END_METHOD

METHOD PRIVATE data2String : BOOL
VAR_INPUT
END_VAR
VAR
	i:UDINT:=0;
END_VAR
//judge length
IF gMAX_CSV_ROWS<(gMAX_BOOL_NUM+gMAX_DINT_NUM+gMAX_LREAL_NUM+3) THEN
	error:=TRUE;
	errTxt:='dataBase$'s length too short';
	RETURN;
END_IF
IF csv_rows<(dataBoolLength+dataDintLength+dataLrealLength+3) THEN
	error:=TRUE;
	errTxt:='dataBase$'s length too short';
	RETURN;
END_IF


//bool
FOR i:=0 TO dataBoolLength DO
	pDatabase[i+1,0]:=TO_STRING(i);//num
	pDatabase[i+1,1]:='BOOL';//data type
	pDatabase[i+1,2]:=TO_STRING(i);;//name
	pDatabase[i+1,3]:=TO_STRING(dataBool[i]);//value
	pDatabase[i+1,4]:='';//no use
END_FOR

//dint
FOR i:=(dataBoolLength+1) TO (dataBoolLength+1+dataDintLength) DO
	pDatabase[i+1,0]:=TO_STRING(i);//num
	pDatabase[i+1,1]:='DINT';//data type
	pDatabase[i+1,2]:=TO_STRING(i-(dataBoolLength+1));;//name
	pDatabase[i+1,3]:=TO_STRING(dataDint[i-(dataBoolLength+1)]);//value
	pDatabase[i+1,4]:='';//no use
END_FOR

//lreal
FOR i:=(dataBoolLength+dataDintLength+2) TO (dataBoolLength+dataDintLength+dataLrealLength+2) DO
	pDatabase[i+1,0]:=TO_STRING(i);//num
	pDatabase[i+1,1]:='LREAL';//data type
	pDatabase[i+1,2]:=TO_STRING(i-(dataBoolLength+dataDintLength+2));;//name
	pDatabase[i+1,3]:=TO_STRING(dataLreal[i-(dataBoolLength+dataDintLength+2)]);//value
	pDatabase[i+1,4]:='';//no use
END_FOR
END_METHOD

METHOD getBoolValue : BOOL
VAR_IN_OUT
	value:BOOL;
END_VAR
VAR_INPUT
	num:UDINT;
END_VAR
IF 0<=num AND num<=dataBoolLength THEN
	value:=dataBool[num];
	getBoolValue:=TRUE;
ELSE
	value:=FALSE;
	getBoolValue:=FALSE;
END_IF
END_METHOD

METHOD getDintValue : BOOL
VAR_IN_OUT
	value:DINT;
END_VAR
VAR_INPUT
	num:UDINT;
END_VAR
IF 0<=num AND num<=dataDintLength THEN
	value:=dataDint[num];
	getDintValue:=TRUE;
ELSE
	value:=0;
	getDintValue:=FALSE;
END_IF
END_METHOD

METHOD getLrealValue : BOOL
VAR_IN_OUT
	value:LREAL;
END_VAR
VAR_INPUT
	num:UDINT;
END_VAR
IF 0<=num AND num<=dataLrealLength THEN
	value:=dataLreal[num];
	getLrealValue:=TRUE;
ELSE
	value:=0;
	getLrealValue:=FALSE;
END_IF
END_METHOD

METHOD PRIVATE getSystemTime : BOOL
VAR_INPUT
END_VAR
//获取本地系统时间--输出到变量 systemTIMEStr
CASE getSystemTimeStep OF
0:
	ntGetTime(
		NETID:= , 
		START:= FALSE, 
		TMOUT:= , 
		BUSY=> , 
		ERR=> , 
		ERRID=> , 
		TIMESTR=> systemTimeStruct);
	IF NOT ntGetTime.BUSY AND NOT ntGetTime.ERR THEN
		getSystemTimeStep:=getSystemTimeStep+1;
	END_IF
1:
	ntGetTime(
		NETID:= , 
		START:= TRUE, 
		TMOUT:= , 
		BUSY=> , 
		ERR=> , 
		ERRID=> , 
		TIMESTR=> systemTimeStruct);
	IF NOT ntGetTime.BUSY AND NOT ntGetTime.ERR THEN
		systemTIMEStr:=SYSTEMTIME_TO_STRING(systemTimeStruct);//系统时间转成字符串格式
		
		sysTIMEStrYY:=WORD_TO_DECSTR(in:=systemTimeStruct.wYear,iPrecision:=4);
		sysTIMEStrMM:=WORD_TO_DECSTR(in:=systemTimeStruct.wMonth,iPrecision:=2);
		sysTIMEStrDD:=WORD_TO_DECSTR(in:=systemTimeStruct.wDay,iPrecision:=2);
		sysTIMEStr_HH:=WORD_TO_DECSTR(in:=systemTimeStruct.wHour,iPrecision:=2);
		sysTIMEStr_mm:=WORD_TO_DECSTR(in:=systemTimeStruct.wMinute,iPrecision:=2);
		sysTIMEStr_ss:=WORD_TO_DECSTR(in:=systemTimeStruct.wSecond,iPrecision:=2);
		
		systemTIMEStr2:='';
		systemTIMEStr2:=CONCAT(systemTIMEStr2,sysTIMEStrYY);
		systemTIMEStr2:=CONCAT(systemTIMEStr2,sysTIMEStrMM);
		systemTIMEStr2:=CONCAT(systemTIMEStr2,sysTIMEStrDD);
		systemTIMEStr2:=CONCAT(systemTIMEStr2,sysTIMEStr_HH);
		systemTIMEStr2:=CONCAT(systemTIMEStr2,sysTIMEStr_mm);
		systemTIMEStr2:=CONCAT(systemTIMEStr2,sysTIMEStr_ss);
		
		getSystemTimeStep:=0;
	ELSIF ntGetTime.ERR THEN
		systemTIMEStr:='';
		getSystemTimeStep:=0;
	END_IF	
END_CASE
END_METHOD

METHOD PRIVATE init : BOOL
VAR_INPUT
END_VAR
VAR
	i:UDINT:=0;
END_VAR
//创建生成初始表格
//judge length
IF gMAX_CSV_ROWS<(gMAX_BOOL_NUM+gMAX_DINT_NUM+gMAX_LREAL_NUM+3) THEN
	error:=TRUE;
	errTxt:='dataBase$'s length too short';
	RETURN;
END_IF
IF csv_rows<(dataBoolLength+dataDintLength+dataLrealLength+3) THEN
	error:=TRUE;
	errTxt:='dataBase$'s length too short';
	RETURN;
END_IF


IF initB AND (NOT busy) THEN
	RETURN;
END_IF
initB:=TRUE;

//header
	pDatabase[0,0]:='NUM';//NUM
	pDatabase[0,1]:='DATA_TYPE';//data type
	pDatabase[0,2]:='NAME';//name
	pDatabase[0,3]:='VALUE';//value
	pDatabase[0,4]:='NO USE';//no use
(*--- 不在此处填充，转移到保存数据时填充
//bool
FOR i:=1 TO (dataBoolLength+1) DO
	//pDatabase[i,0]:=UDINT_TO_STRING(i-1);//NUM  --- 不在此处填充
	//pDatabase[i,1]:='BOOL';//data type --- 不在此处填充
	//pDatabase[i,2]:='';//name
	//pDatabase[i,3]:=BOOL_TO_STRING(FALSE);//value
	//pDatabase[i,4]:='';//no use
END_FOR

//dint
FOR i:=(dataBoolLength+2) TO (dataBoolLength+2+dataDintLength) DO
	//pDatabase[i,0]:=UDINT_TO_STRING(i-(dataBoolLength+2));//NUM  --- 不在此处填充
	//pDatabase[i,1]:='DINT';//data type --- 不在此处填充
	//pDatabase[i,2]:='';//name
	//pDatabase[i,3]:=DINT_TO_STRING(0);//value
	//pDatabase[i,4]:='';//no use
END_FOR

//lreal
FOR i:=(dataBoolLength+dataDintLength+3) TO (dataBoolLength+dataDintLength+dataLrealLength+3) DO
	//pDatabase[i,0]:=UDINT_TO_STRING(i-(dataBoolLength+dataDintLength+3));//NUM  --- 不在此处填充
	//pDatabase[i,1]:='LREAL';//data type --- 不在此处填充
	//pDatabase[i,2]:='';//name
	//pDatabase[i,3]:=DINT_TO_STRING(0);//value
	//pDatabase[i,4]:='';//no use
END_FOR
*)
END_METHOD

METHOD PRIVATE readMethod : BOOL
VAR_INPUT
END_VAR
CASE readStep OF
0:
	IF (readB OR (NOT startUPb)) AND (NOT busy) THEN
		readStep:=1;
		startUPb:=TRUE;//for first time, 
		readB:=FALSE;
		rDone:=FALSE;
		busy:=TRUE;
		error:=FALSE;
		errID:=0;
		errTxt:='';
		fbFileOpen(bExecute:= FALSE);
		checkFileExistError:=FALSE;
	END_IF
	
1:
	fbFileOpen(
		sNetId:= , 
		sPathName:= sFileName, 
		nMode:= FOPEN_MODEREAD, 
		ePath:= PATH_GENERIC, 
		bExecute:= TRUE, 
		tTimeout:= , 
		bBusy=> , 
		bError=> , 
		nErrId=> , 
		hFile=> hFile);
	IF NOT fbFileOpen.bBusy THEN
		IF fbFileOpen.bError THEN
			checkFileExistError:=TRUE;
		END_IF
		fbFileOpen(bExecute:= FALSE);
		readStep:=2;
	END_IF
	fbFileClose(bExecute:= FALSE);
2:
	fbFileClose(
		sNetId:= , 
		hFile:= hFile, 
		bExecute:= TRUE, 
		tTimeout:= , 
		bBusy=> , 
		bError=> , 
		nErrId=> );
	IF NOT fbFileClose.bBusy THEN
		IF checkFileExistError THEN
			readStep:=110;
		ELSE
			readStep:=11;
		END_IF
		fbFileClose(bExecute:= FALSE);
	END_IF

11:
	//read txt to Database
	readTxt(
		database:= pDatabase, 
		csv_rows:= csv_rows, 
		csv_columns:= csv_columns, 
		bRead:= TRUE, 
		sFileName:= sFileName);
	readStep:=12;

12:
	readTxt(
		database:= pDatabase, 
		csv_rows:= csv_rows, 
		csv_columns:= csv_columns, 
		bRead:= FALSE, 
		sFileName:= sFileName,
		Error=>error,
		nErrId=>errID);
		
	IF error THEN
		readStep:=110;
		RETURN;
	END_IF
	
	IF NOT readTxt.bBusy THEN
		readStep:=13;
	END_IF
	
13:
	string2Data();
	readStep:=100;
	
100:
	rDone:=TRUE;
	busy:=FALSE;
	error:=error;
	errID:=errID;
	errTxt:=errTxt;
	IF NOT readB THEN
		readStep:=0;
	END_IF	


110:
	rDone:=FALSE;
	busy:=FALSE;
	error:=TRUE;
	errID:=errID;
	errTxt:='read data fail';	
	IF NOT readB THEN
		readStep:=0;
	END_IF		
	
END_CASE
END_METHOD

METHOD PRIVATE saveMethod : BOOL
VAR_INPUT
END_VAR
CASE saveStep OF
0:
	IF saveB AND (NOT busy) THEN
		saveStep:=1;
		saveB:=FALSE;
		busy:=TRUE;
		sDone:=FALSE;
		error:=FALSE;
		errID:=0;
		errTxt:='';
	END_IF

1:
	createDir();
	data2String();
	saveStep:=2;

2:
	writeTxt(
		database:= pDatabase, 
		csv_rows:= csv_rows, 
		csv_columns:= csv_columns, 
		bWrite:= TRUE, 
		sFileName:= sFileName,
		sFileNameOld:= sFileNameOld);	
	saveStep:=3;

3:
	writeTxt(
		database:= pDatabase, 
		csv_rows:= csv_rows, 
		csv_columns:= csv_columns, 
		bWrite:= FALSE, 
		sFileName:= sFileName,
		sFileNameOld:= sFileNameOld,
		Error=>error,
		nErrID=>errID);	
	
	IF error THEN
		saveStep:=110;
		RETURN;
	END_IF

	IF NOT writeTxt.bBusy THEN
		saveStep:=100;
	END_IF

100:
	busy:=FALSE;
	sDone:=TRUE;
	error:=error;
	errID:=errID;
	errTxt:=errTxt;

	IF NOT saveB THEN
		saveStep:=0;
	END_IF

110:
	busy:=FALSE;
	sDone:=FALSE;
	error:=TRUE;
	errID:=errID;
	errTxt:='save data fail';

	IF NOT saveB THEN
		saveStep:=0;
	END_IF
END_CASE
END_METHOD

METHOD setBoolValue : BOOL
VAR_INPUT
	value:BOOL;
END_VAR
VAR_INPUT
	num:UDINT;
END_VAR
IF 0<=num AND num<=dataBoolLength THEN
	dataBool[num]:=value;
	setBoolValue:=TRUE;
ELSE
	setBoolValue:=FALSE;
END_IF
END_METHOD

METHOD setDintValue : BOOL
VAR_INPUT
	value:DINT;
END_VAR
VAR_INPUT
	num:UDINT;
END_VAR
IF 0<=num AND num<=dataDintLength THEN
	dataDint[num]:=value;
	setDintValue:=TRUE;
ELSE
	setDintValue:=FALSE;
END_IF
END_METHOD

METHOD setLrealValue : BOOL
VAR_INPUT
	value:LREAL;
END_VAR
VAR_INPUT
	num:UDINT;
END_VAR

IF 0<=num AND num<=dataLrealLength THEN
	dataLreal[num]:=value;
	setLrealValue:=TRUE;
ELSE
	setLrealValue:=FALSE;
END_IF
END_METHOD

METHOD PRIVATE string2Data : BOOL
VAR_INPUT
END_VAR
VAR
	i:UDINT:=0;
	index_temp:UDINT;
END_VAR
//judge length
IF gMAX_CSV_ROWS<(gMAX_BOOL_NUM+gMAX_DINT_NUM+gMAX_LREAL_NUM+3) THEN
	error:=TRUE;
	errTxt:='dataBase$'s length too short';
	RETURN;
END_IF
IF csv_rows<(dataBoolLength+dataDintLength+dataLrealLength+3) THEN
	error:=TRUE;
	errTxt:='dataBase$'s length too short';
	RETURN;
END_IF

(*
//bool
FOR i:=0 TO dataBoolLength DO
	dataBool[i]:=STRING_TO_BOOL(pDatabase[i+1,3]);//value
END_FOR

//dint
FOR i:=(dataBoolLength+1) TO (dataBoolLength+1+dataDintLength) DO
	dataDint[i-(dataBoolLength+1)]:=STRING_TO_DINT(pDatabase[i+1,3]);//value
END_FOR

//lreal
FOR i:=(dataBoolLength+dataDintLength+2) TO (dataBoolLength+dataDintLength+dataLrealLength+2) DO
	dataLreal[i-(dataBoolLength+dataDintLength+2)]:=STRING_TO_LREAL(pDatabase[i+1,3]);//value
END_FOR
*)
FOR i:=0 TO gMAX_CSV_ROWS DO
	index_temp:=TO_UDINT(pDatabase[i,2]);
	
	IF 'BOOL'=pDatabase[i,1] 
		AND 0<=index_temp  
		AND index_temp<=dataBoolLength THEN
		dataBool[index_temp]:=TO_BOOL(pDatabase[i,3]);
	END_IF
	IF 'DINT'=pDatabase[i,1] 
		AND 0<=index_temp  
		AND index_temp<=dataDintLength THEN
		dataDint[index_temp]:=TO_DINT(pDatabase[i,3]);
	END_IF
	IF 'LREAL'=pDatabase[i,1] 
		AND 0<=index_temp  
		AND index_temp<=dataLrealLength THEN
		dataLreal[index_temp]:=TO_LREAL(pDatabase[i,3]);
	END_IF
END_FOR
END_METHOD

ACTION VersionLog:
(*
版本: V1.0.0.0
说明:
	1. 首个版本
(**************************************************)
版本: V1.0.0.1
说明:
	1. 增加参数备份文件，文件名以原文件名+时间命名
(**************************************************)
*)
END_ACTION

END_FUNCTION_BLOCK

// ---- POUs/BaseModule/DataSaveModule_EX/csvReadWriteInTextMode/P_TextModeWrite.TcPOU
FUNCTION_BLOCK P_TextModeWrite
VAR_IN_OUT
	database		: ARRAY[0..gMAX_CSV_ROWS, 0..gMAX_CSV_COLUMNS ] OF STRING(30);
	csv_rows		: UDINT;
	csv_columns		: UDINT;
END_VAR
VAR_INPUT
	bWrite			: BOOL := FALSE;(* Rising edge starts program execution *)	
	sFileName		: T_MaxString := '';(* CSV destination file path and name *)
	sFileNameOld	:T_MaxString := '';(*旧文件名*)
END_VAR
VAR_OUTPUT
	bBusy			: BOOL;
	error			: BOOL;
	nErrId			: UDINT;	
END_VAR
VAR
	bError			: BOOL;
	sNetId			: T_AmsNetId := '';	(* TwinCAT system network address *)

